KUKA KRL program: MyProgram_093().src

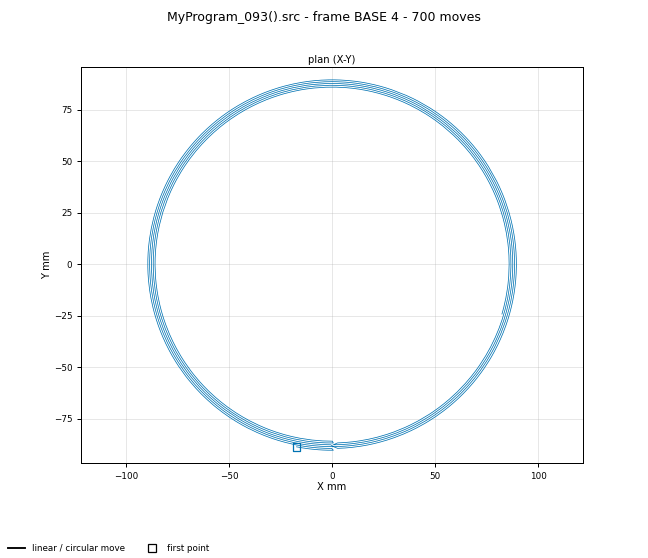
[picture p0: tool path of MyProgram_093().src in frame BASE 4, 700 of 700 moves have a stored position in this frame; points joined in program order, loops and branches not executed]
&ACCESS RVP
&REL 1
&PARAM TEMPLATE = C:\KRC\Roboter\Template\vorgabe
&PARAM EDITMASK = *
DEF MyProgram_093()
; ---- Setting reference (Base) ----
$BASE = BASE_DATA[4]

; --------------------------
; ---- Setting tool (TCP) ----
$TOOL = TOOL_DATA[3]
; --------------------------

$VEL.CP = VEL_APROX_PRINT
Startdeposition()
$VEL.CP = VEL_PRINT
LIN {X -17.2677,Y -88.7195,Z 88,A -105.0819,B 24.9302,C -1.9284,E1 24.9711,E2 190.1577} C_DIS
LIN {X -14.1349,Y -89.2726,Z 88,A -103.3335,B 24.931,C -1.9189,E1 24.9759,E2 188.4301} C_DIS
LIN {X -11.9398,Y -89.5926,Z 88,A -101.7935,B 24.9307,C -1.923,E1 24.9801,E2 186.8791} C_DIS
LIN {X -9.7374,Y -89.8586,Z 88,A -100.3354,B 24.9306,C -1.9245,E1 24.9842,E2 185.4164} C_DIS
LIN {X -6.6492,Y -90.1409,Z 88,A -98.31,B 24.9304,C -1.9264,E1 24.9899,E2 183.3856} C_DIS
LIN {X -4.435,Y -90.2769,Z 88,A -96.9041,B 24.9304,C -1.9265,E1 24.9938,E2 181.9792} C_DIS
LIN {X -2.2182,Y -90.3586,Z 88,A -95.6086,B 24.9307,C -1.923,E1 24.9974,E2 180.6918} C_DIS
LIN {X 0.6077,Y -90.3807,Z 88,A -93.9914,B 24.9311,C -1.9176,E1 25.0019,E2 179.0874} C_DIS
Enddeposition()
LIN {X 0.6077,Y -90.3807,Z 88,A -93.9914,B 24.9311,C -1.9176,E1 25.0019,E2 179.0874} C_DIS
Startdeposition()
$VEL.CP = VEL_PRINT
LIN {X -0.2018,Y -89.5034,Z 88,A -95.2008,B 24.9316,C -1.91,E1 24.9984,E2 180.3149} C_DIS
LIN {X -3.7428,Y -89.4247,Z 88,A -97.2969,B 24.9312,C -1.9153,E1 24.9926,E2 182.3987} C_DIS
LIN {X -6.611,Y -89.26,Z 88,A -99.3502,B 24.9317,C -1.9083,E1 24.9868,E2 184.4693} C_DIS
LIN {X -9.99,Y -88.9447,Z 88,A -101.4992,B 24.9317,C -1.9092,E1 24.9809,E2 186.6173} C_DIS
LIN {X -13.5317,Y -88.4743,Z 88,A -103.6581,B 24.9313,C -1.9139,E1 24.9749,E2 188.7669} C_DIS
LIN {X -16.6632,Y -87.9386,Z 88,A -105.8021,B 24.9315,C -1.911,E1 24.969,E2 190.9198} C_DIS
LIN {X -19.0714,Y -87.4475,Z 88,A -107.3659,B 24.9315,C -1.912,E1 24.9647,E2 192.4831} C_DIS
LIN {X -22.7883,Y -86.5549,Z 88,A -109.8141,B 24.9314,C -1.9133,E1 24.9581,E2 194.9317} C_DIS
LIN {X -26.1366,Y -85.6026,Z 88,A -112.07,B 24.9314,C -1.914,E1 24.9521,E2 197.1898} C_DIS
LIN {X -29.0903,Y -84.6452,Z 88,A -114.4014,B 24.932,C -1.9048,E1 24.9458,E2 199.5475} C_DIS
LIN {X -32.8513,Y -83.2562,Z 88,A -116.3989,B 24.9305,C -1.925,E1 24.9407,E2 201.501} C_DIS
LIN {X -36.4844,Y -81.7299,Z 88,A -119.5254,B 24.9317,C -1.9088,E1 24.9326,E2 204.6734} C_DIS
LIN {X -40.9536,Y -79.5842,Z 88,A -122.2051,B 24.9303,C -1.928,E1 24.926,E2 207.3145} C_DIS
LIN {X -43.6945,Y -78.1126,Z 88,A -124.3723,B 24.9305,C -1.9253,E1 24.9206,E2 209.4945} C_DIS
LIN {X -46.616,Y -76.4052,Z 88,A -126.2873,B 24.9297,C -1.9361,E1 24.9161,E2 211.3894} C_DIS
LIN {X -50.1403,Y -74.14,Z 88,A -129.7875,B 24.9312,C -1.9153,E1 24.9078,E2 214.9507} C_DIS
LIN {X -53.1864,Y -71.9871,Z 88,A -131.414,B 24.9293,C -1.9425,E1 24.9043,E2 216.5181} C_DIS
LIN {X -55.7787,Y -69.9975,Z 88,A -133.5713,B 24.9291,C -1.9443,E1 24.8995,E2 218.6792} C_DIS
LIN {X -57.6179,Y -68.4926,Z 88,A -135.3866,B 24.9296,C -1.9382,E1 24.8956,E2 220.5159} C_DIS
LIN {X -60.6071,Y -65.8603,Z 88,A -137.8417,B 24.929,C -1.9461,E1 24.8905,E2 222.962} C_DIS
LIN {X -63.6381,Y -62.9364,Z 88,A -140.4239,B 24.9283,C -1.9551,E1 24.8854,E2 225.5335} C_DIS
LIN {X -65.9632,Y -60.495,Z 88,A -142.6569,B 24.9282,C -1.9576,E1 24.8811,E2 227.7704} C_DIS
LIN {X -69.4849,Y -56.4149,Z 88,A -146.0739,B 24.9275,C -1.9665,E1 24.8749,E2 231.1817} C_DIS
LIN {X -71.1283,Y -54.3295,Z 88,A -147.9693,B 24.9276,C -1.9647,E1 24.8717,E2 233.0904} C_DIS
LIN {X -74.4966,Y -49.6106,Z 88,A -151.3869,B 24.9263,C -1.9827,E1 24.8663,E2 236.4819} C_DIS
LIN {X -75.9809,Y -47.3044,Z 88,A -153.3686,B 24.9265,C -1.9806,E1 24.8633,E2 238.4788} C_DIS
LIN {X -77.7777,Y -44.2893,Z 88,A -155.6267,B 24.926,C -1.9862,E1 24.8601,E2 240.7353} C_DIS
LIN {X -79.0548,Y -41.9667,Z 88,A -157.3694,B 24.9258,C -1.9894,E1 24.8578,E2 242.4794} C_DIS
LIN {X -80.6854,Y -38.7382,Z 88,A -159.5317,B 24.925,C -2.0004,E1 24.8551,E2 244.6274} C_DIS
LIN {X -82.1108,Y -35.6177,Z 88,A -161.8296,B 24.9247,C -2.0036,E1 24.8525,E2 246.9302} C_DIS
LIN {X -83.3917,Y -32.5064,Z 88,A -164.0572,B 24.9244,C -2.0077,E1 24.8502,E2 249.1605} C_DIS
LIN {X -84.4231,Y -29.7244,Z 88,A -165.8189,B 24.9237,C -2.0172,E1 24.8485,E2 250.9093} C_DIS
LIN {X -85.4184,Y -26.7309,Z 88,A -167.9478,B 24.9235,C -2.0201,E1 24.8467,E2 253.0437} C_DIS
LIN {X -86.2514,Y -23.9112,Z 88,A -169.6906,B 24.9227,C -2.0298,E1 24.8454,E2 254.7735} C_DIS
LIN {X -86.9893,Y -21.0635,Z 88,A -171.7604,B 24.9227,C -2.0301,E1 24.844,E2 256.8545} C_DIS
LIN {X -88.0046,Y -16.3156,Z 88,A -174.9311,B 24.9221,C -2.0379,E1 24.8422,E2 260.0254} C_DIS
LIN {X -88.5955,Y -12.7139,Z 88,A -177.5639,B 24.9222,C -2.0367,E1 24.8411,E2 262.6767} C_DIS
LIN {X -89.16,Y -7.8382,Z 88,A 179.5846,B 24.9208,C -2.0549,E1 24.8403,E2 265.5017} C_DIS
LIN {X -89.3876,Y -4.5587,Z 88,A 177.4493,B 24.9204,C -2.0607,E1 24.8399,E2 267.636} C_DIS
LIN {X -89.4911,Y -1.4707,Z 88,A 175.3618,B 24.9201,C -2.0639,E1 24.8398,E2 269.7285} C_DIS
LIN {X -89.4749,Y 2.2886,Z 88,A 173.034,B 24.9193,C -2.0738,E1 24.8398,E2 272.0467} C_DIS
LIN {X -89.3176,Y 5.7646,Z 88,A 170.7534,B 24.9189,C -2.0795,E1 24.8402,E2 274.3276} C_DIS
LIN {X -89.0787,Y 8.7189,Z 88,A 168.9357,B 24.9183,C -2.0878,E1 24.8407,E2 276.1363} C_DIS
LIN {X -88.6731,Y 12.1676,Z 88,A 165.5912,B 24.9202,C -2.063,E1 24.842,E2 279.5599} C_DIS
LIN {X -87.7877,Y 17.4455,Z 88,A 163.4378,B 24.9165,C -2.1101,E1 24.8431,E2 281.6135} C_DIS
LIN {X -86.6183,Y 22.5416,Z 88,A 159.8021,B 24.9163,C -2.1124,E1 24.8454,E2 285.2653} C_DIS
LIN {X -85.642,Y 26.0098,Z 88,A 157.6135,B 24.9155,C -2.123,E1 24.8471,E2 287.4412} C_DIS
LIN {X -84.9077,Y 28.3119,Z 88,A 155.9613,B 24.9153,C -2.1247,E1 24.8485,E2 289.0986} C_DIS
LIN {X -83.7002,Y 31.7028,Z 88,A 153.6656,B 24.9147,C -2.1321,E1 24.8507,E2 291.3899} C_DIS
LIN {X -82.4438,Y 34.8398,Z 88,A 151.4698,B 24.9143,C -2.1377,E1 24.8531,E2 293.5845} C_DIS
LIN {X -81.0499,Y 37.9703,Z 88,A 149.4534,B 24.9134,C -2.1494,E1 24.8554,E2 295.5839} C_DIS
LIN {X -79.8135,Y 40.5051,Z 88,A 147.599,B 24.913,C -2.1533,E1 24.8577,E2 297.439} C_DIS
LIN {X -78.7808,Y 42.4785,Z 88,A 145.6712,B 24.9139,C -2.1429,E1 24.8603,E2 299.4018} C_DIS
LIN {X -76.5712,Y 46.3429,Z 88,A 143.1007,B 24.9126,C -2.1591,E1 24.8639,E2 301.9469} C_DIS
LIN {X -74.7509,Y 49.2249,Z 88,A 141.0808,B 24.9117,C -2.1699,E1 24.8669,E2 303.9513} C_DIS
LIN {X -72.9491,Y 51.8579,Z 88,A 139.0218,B 24.9113,C -2.175,E1 24.8702,E2 306.0082} C_DIS
LIN {X -70.896,Y 54.631,Z 88,A 136.746,B 24.9109,C -2.179,E1 24.874,E2 308.2855} C_DIS
LIN {X -68.7971,Y 57.2516,Z 88,A 134.6193,B 24.9104,C -2.1852,E1 24.8777,E2 310.4072} C_DIS
LIN {X -66.6997,Y 59.6819,Z 88,A 132.4938,B 24.9102,C -2.1884,E1 24.8817,E2 312.5348} C_DIS
LIN {X -64.9308,Y 61.603,Z 88,A 130.9514,B 24.9095,C -2.1963,E1 24.8846,E2 314.0651} C_DIS
LIN {X -63.432,Y 63.145,Z 88,A 128.789,B 24.9111,C -2.1766,E1 24.889,E2 316.2837} C_DIS
LIN {X -60.7666,Y 65.714,Z 88,A 127.0312,B 24.9092,C -2.2,E1 24.8924,E2 317.9927} C_DIS
LIN {X -58.1889,Y 68.0064,Z 88,A 124.7992,B 24.9089,C -2.2043,E1 24.8971,E2 320.2233} C_DIS
LIN {X -55.9485,Y 69.8629,Z 88,A 122.8516,B 24.9087,C -2.2058,E1 24.9014,E2 322.1746} C_DIS
LIN {X -53.4359,Y 71.8021,Z 88,A 120.9029,B 24.9082,C -2.2125,E1 24.9057,E2 324.1144} C_DIS
LIN {X -50.8147,Y 73.6801,Z 88,A 118.8448,B 24.9078,C -2.2168,E1 24.9104,E2 326.1693} C_DIS
LIN {X -48.2042,Y 75.4133,Z 88,A 116.8196,B 24.9075,C -2.2201,E1 24.9151,E2 328.1933} C_DIS
LIN {X -45.5838,Y 77.0253,Z 88,A 114.7982,B 24.9074,C -2.2221,E1 24.9199,E2 330.2161} C_DIS
LIN {X -42.1374,Y 78.9649,Z 88,A 111.5734,B 24.9087,C -2.2056,E1 24.928,E2 333.4893} C_DIS
LIN {X -38.5937,Y 80.7549,Z 88,A 109.2049,B 24.908,C -2.2148,E1 24.9339,E2 335.8421} C_DIS
LIN {X -35.4902,Y 82.166,Z 88,A 107.6558,B 24.9061,C -2.2371,E1 24.9377,E2 337.3416} C_DIS
LIN {X -32.6192,Y 83.3474,Z 88,A 105.4788,B 24.9064,C -2.2341,E1 24.9434,E2 339.5308} C_DIS
LIN {X -29.7668,Y 84.4082,Z 88,A 103.7025,B 24.9057,C -2.2418,E1 24.948,E2 341.2922} C_DIS
LIN {X -25.866,Y 85.685,Z 88,A 100.9377,B 24.9058,C -2.2406,E1 24.9554,E2 344.0648} C_DIS
LIN {X -23.2236,Y 86.4376,Z 88,A 98.3447,B 24.9078,C -2.2168,E1 24.9626,E2 346.7182} C_DIS
LIN {X -18.8337,Y 87.4993,Z 88,A 96.2593,B 24.9055,C -2.2442,E1 24.9681,E2 348.7413} C_DIS
LIN {X -14.431,Y 88.3326,Z 88,A 93.5704,B 24.9049,C -2.252,E1 24.9754,E2 351.4145} C_DIS
LIN {X -11.5589,Y 88.7535,Z 88,A 91.666,B 24.9049,C -2.2517,E1 24.9807,E2 353.3209} C_DIS
LIN {X -8.7008,Y 89.0803,Z 88,A 89.6908,B 24.9052,C -2.2484,E1 24.9862,E2 355.305} C_DIS
LIN {X -5.2715,Y 89.3482,Z 88,A 87.4703,B 24.9052,C -2.2488,E1 24.9924,E2 357.5256} C_DIS
LIN {X -1.6513,Y 89.4878,Z 88,A 85.3192,B 24.9046,C -2.2548,E1 24.9984,E2 359.6628} C_DIS
LIN {X 1.2208,Y 89.4957,Z 88,A 83.5226,B 24.9045,C -2.2565,E1 25.0034,E2 361.4553} C_DIS
LIN {X 3.9685,Y 89.415,Z 88,A 81.5419,B 24.9051,C -2.2496,E1 25.0089,E2 363.4518} C_DIS
LIN {X 7.649,Y 89.177,Z 88,A 79.1414,B 24.9051,C -2.2482,E1 25.0156,E2 365.8545} C_DIS
LIN {X 11.3103,Y 88.7857,Z 88,A 76.8921,B 24.9049,C -2.2512,E1 25.0218,E2 368.0948} C_DIS
LIN {X 14.1032,Y 88.3859,Z 88,A 75.0274,B 24.9051,C -2.2488,E1 25.027,E2 369.9635} C_DIS
LIN {X 16.6245,Y 87.946,Z 88,A 73.3814,B 24.9052,C -2.2479,E1 25.0315,E2 371.6098} C_DIS
LIN {X 20.2306,Y 87.1867,Z 88,A 71.1863,B 24.9049,C -2.2521,E1 25.0375,E2 373.792} C_DIS
LIN {X 22.8843,Y 86.5293,Z 88,A 69.2148,B 24.9056,C -2.2438,E1 25.0429,E2 375.7802} C_DIS
LIN {X 25.8223,Y 85.698,Z 88,A 66.9153,B 24.9066,C -2.2311,E1 25.0491,E2 378.1057} C_DIS
LIN {X 28.8694,Y 84.7197,Z 88,A 65.256,B 24.9057,C -2.2422,E1 25.0534,E2 379.7357} C_DIS
LIN {X 36.0471,Y 81.9237,Z 88,A 60.3436,B 24.9061,C -2.2378,E1 25.0661,E2 384.6473} C_DIS
LIN {X 39.2906,Y 80.4195,Z 88,A 58.3164,B 24.9056,C -2.2438,E1 25.0712,E2 386.6551} C_DIS
LIN {X 41.6313,Y 79.2315,Z 88,A 56.109,B 24.9072,C -2.2241,E1 25.0767,E2 388.903} C_DIS
LIN {X 47.5385,Y 75.8347,Z 88,A 51.4751,B 24.9085,C -2.2086,E1 25.0879,E2 393.5592} C_DIS
LIN {X 50.7352,Y 73.7354,Z 88,A 49.6306,B 24.9071,C -2.2248,E1 25.0921,E2 395.359} C_DIS
LIN {X 53.557,Y 71.7112,Z 88,A 47.4868,B 24.9072,C -2.2237,E1 25.0969,E2 397.4979} C_DIS
LIN {X 55.8435,Y 69.9463,Z 88,A 45.6499,B 24.9075,C -2.2207,E1 25.1009,E2 399.3351} C_DIS
LIN {X 57.7632,Y 68.3691,Z 88,A 44.2922,B 24.9071,C -2.2257,E1 25.1038,E2 400.6759} C_DIS
LIN {X 60.1768,Y 66.2551,Z 88,A 41.9475,B 24.9082,C -2.2117,E1 25.1087,E2 403.0443} C_DIS
LIN {X 62.7183,Y 63.8534,Z 88,A 39.7767,B 24.9084,C -2.2094,E1 25.1131,E2 405.2116} C_DIS
LIN {X 64.9615,Y 61.5703,Z 88,A 37.6939,B 24.9089,C -2.2038,E1 25.1171,E2 407.2987} C_DIS
LIN {X 66.5632,Y 59.8344,Z 88,A 36.1594,B 24.9092,C -2.1996,E1 25.12,E2 408.8362} C_DIS
LIN {X 68.486,Y 57.6259,Z 88,A 34.2585,B 24.9097,C -2.1944,E1 25.1235,E2 410.7408} C_DIS
LIN {X 70.6649,Y 54.9308,Z 88,A 32.1916,B 24.9097,C -2.1944,E1 25.127,E2 412.7981} C_DIS
LIN {X 72.0544,Y 53.0944,Z 88,A 30.6065,B 24.9103,C -2.1869,E1 25.1297,E2 414.3932} C_DIS
LIN {X 74.1876,Y 50.07,Z 88,A 28.4301,B 24.9103,C -2.1877,E1 25.1331,E2 416.5571} C_DIS
LIN {X 75.8828,Y 47.4615,Z 88,A 26.1245,B 24.9115,C -2.1716,E1 25.1366,E2 418.8891} C_DIS
LIN {X 79.9299,Y 40.2772,Z 88,A 21.0065,B 24.9123,C -2.1629,E1 25.1435,E2 424.0009} C_DIS
LIN {X 81.5034,Y 36.9869,Z 88,A 18.785,B 24.9125,C -2.1603,E1 25.1461,E2 426.2164} C_DIS
LIN {X 82.8611,Y 33.8353,Z 88,A 16.686,B 24.9127,C -2.1575,E1 25.1484,E2 428.3106} C_DIS
LIN {X 84.0143,Y 30.8614,Z 88,A 14.3901,B 24.9139,C -2.1425,E1 25.1507,E2 430.629} C_DIS
LIN {X 85.8827,Y 25.1996,Z 88,A 10.5558,B 24.9149,C -2.1305,E1 25.1539,E2 434.4699} C_DIS
LIN {X 86.8929,Y 21.4584,Z 88,A 8.2472,B 24.9149,C -2.129,E1 25.1555,E2 436.7687} C_DIS
LIN {X 87.6431,Y 18.1519,Z 88,A 6.0741,B 24.9155,C -2.1223,E1 25.1568,E2 438.9451} C_DIS
LIN {X 88.3202,Y 14.5052,Z 88,A 3.9319,B 24.9155,C -2.1231,E1 25.1578,E2 441.0728} C_DIS
LIN {X 88.737,Y 11.6858,Z 88,A 2.1199,B 24.9159,C -2.1178,E1 25.1585,E2 442.8865} C_DIS
LIN {X 89.062,Y 8.8849,Z 88,A 0.3349,B 24.9163,C -2.1128,E1 25.1591,E2 444.6728} C_DIS
LIN {X 89.31,Y 5.8763,Z 88,A -1.6468,B 24.9169,C -2.1049,E1 25.1595,E2 446.6614} C_DIS
LIN {X 89.4643,Y 2.6332,Z 88,A -3.8473,B 24.9178,C -2.094,E1 25.1598,E2 448.8747} C_DIS
LIN {X 89.4981,Y -1.0756,Z 88,A -6.2174,B 24.9184,C -2.0865,E1 25.1598,E2 451.2484} C_DIS
LIN {X 89.3856,Y -4.5956,Z 88,A -8.4623,B 24.9189,C -2.0796,E1 25.1595,E2 453.4961} C_DIS
LIN {X 89.1712,Y -7.7166,Z 88,A -10.4271,B 24.9193,C -2.0745,E1 25.1591,E2 455.4613} C_DIS
LIN {X 88.8268,Y -10.9927,Z 88,A -12.5395,B 24.9198,C -2.0676,E1 25.1584,E2 457.5775} C_DIS
LIN {X 88.3477,Y -14.3402,Z 88,A -14.7309,B 24.9204,C -2.0597,E1 25.1574,E2 459.7745} C_DIS
LIN {X 87.756,Y -17.6022,Z 88,A -16.4946,B 24.92,C -2.0658,E1 25.1565,E2 461.5136} C_DIS
LIN {X 87.0982,Y -20.6136,Z 88,A -18.7695,B 24.9213,C -2.0487,E1 25.1551,E2 463.8155} C_DIS
LIN {X 86.2975,Y -23.7425,Z 88,A -20.7239,B 24.9215,C -2.0463,E1 25.1537,E2 465.7645} C_DIS
LIN {X 85.4502,Y -26.6282,Z 88,A -22.6821,B 24.922,C -2.0391,E1 25.1521,E2 467.7286} C_DIS
LIN {X 84.4861,Y -29.5448,Z 88,A -24.9873,B 24.9234,C -2.021,E1 25.15,E2 470.0635} C_DIS
LIN {X 83.0641,Y -33.3367,Z 88,A -27.0152,B 24.9225,C -2.033,E1 25.148,E2 472.0517} C_DIS
LIN {X 81.6672,Y -36.6235,Z 88,A -29.3937,B 24.9233,C -2.0228,E1 25.1454,E2 474.4412} C_DIS
LIN {X 80.448,Y -39.2321,Z 88,A -31.4259,B 24.9242,C -2.0106,E1 25.1429,E2 476.4914} C_DIS
LIN {X 78.7402,Y -42.5534,Z 88,A -33.5786,B 24.9241,C -2.0121,E1 25.1401,E2 478.6293} C_DIS
LIN {X 77.4747,Y -44.8165,Z 88,A -35.2901,B 24.9246,C -2.0054,E1 25.1377,E2 480.3476} C_DIS
LIN {X 76.2837,Y -46.8149,Z 88,A -37.6884,B 24.9273,C -1.9692,E1 25.1341,E2 482.8192} C_DIS
LIN {X 73.7357,Y -50.7348,Z 88,A -39.8088,B 24.9256,C -1.9915,E1 25.1309,E2 484.8766} C_DIS
LIN {X 72.3535,Y -52.6859,Z 88,A -41.317,B 24.9259,C -1.9881,E1 25.1284,E2 486.3854} C_DIS
LIN {X 70.2113,Y -55.5082,Z 88,A -43.4754,B 24.9261,C -1.9859,E1 25.1247,E2 488.5388} C_DIS
LIN {X 68.3715,Y -57.7604,Z 88,A -45.5353,B 24.9269,C -1.9741,E1 25.121,E2 490.6172} C_DIS
LIN {X 66.2879,Y -60.1411,Z 88,A -47.5453,B 24.9273,C -1.9695,E1 25.1173,E2 492.6292} C_DIS
LIN {X 63.6878,Y -62.886,Z 88,A -49.7628,B 24.9272,C -1.9706,E1 25.113,E2 494.8343} C_DIS
LIN {X 61.5704,Y -64.9615,Z 88,A -51.7185,B 24.9277,C -1.9641,E1 25.1091,E2 496.7974} C_DIS
LIN {X 59.1043,Y -67.2128,Z 88,A -53.608,B 24.9274,C -1.9678,E1 25.1052,E2 498.6705} C_DIS
LIN {X 56.6616,Y -69.2849,Z 88,A -55.8817,B 24.9283,C -1.9554,E1 25.1003,E2 500.9646} C_DIS
LIN {X 54.0322,Y -71.3542,Z 88,A -58.0083,B 24.9286,C -1.9514,E1 25.0956,E2 503.0931} C_DIS
LIN {X 50.5398,Y -73.8695,Z 88,A -60.7922,B 24.9291,C -1.9448,E1 25.0892,E2 505.8829} C_DIS
LIN {X 47.5934,Y -75.8003,Z 88,A -63.0457,B 24.9294,C -1.9405,E1 25.0839,E2 508.1392} C_DIS
LIN {X 45.0862,Y -77.3189,Z 88,A -65.7477,B 24.9317,C -1.9089,E1 25.0772,E2 510.9076} C_DIS
LIN {X 41.0599,Y -79.5299,Z 88,A -67.8581,B 24.93,C -1.9321,E1 25.0722,E2 512.9572} C_DIS
LIN {X 38.2002,Y -80.9429,Z 88,A -69.9562,B 24.9304,C -1.927,E1 25.0669,E2 515.0621} C_DIS
LIN {X 34.4692,Y -82.6,Z 88,A -72.711,B 24.931,C -1.9183,E1 25.0597,E2 517.8307} C_DIS
LIN {X 30.2241,Y -84.2467,Z 88,A -75.53,B 24.931,C -1.9177,E1 25.0524,E2 520.6453} C_DIS
LIN {X 26.6354,Y -85.448,Z 88,A -77.7297,B 24.9307,C -1.9223,E1 25.0466,E2 522.8299} C_DIS
LIN {X 23.5822,Y -86.3407,Z 88,A -79.7732,B 24.9309,C -1.9198,E1 25.0411,E2 524.876} C_DIS
LIN {X 20.5418,Y -87.1148,Z 88,A -81.8168,B 24.9311,C -1.9166,E1 25.0355,E2 526.9241} C_DIS
LIN {X 17.3379,Y -87.8087,Z 88,A -83.9793,B 24.9314,C -1.9127,E1 25.0296,E2 529.0933} C_DIS
LIN {X 13.9414,Y -88.4109,Z 88,A -86.2356,B 24.9317,C -1.9094,E1 25.0234,E2 531.355} C_DIS
LIN {X 9.9536,Y -88.949,Z 88,A -88.7751,B 24.9317,C -1.909,E1 25.0163,E2 533.8935} C_DIS
LIN {X 6.3255,Y -89.2797,Z 88,A -91.0284,B 24.9316,C -1.9105,E1 25.0101,E2 536.1421} C_DIS
LIN {X 2.7078,Y -89.462,Z 88,A -93.338,B 24.9316,C -1.91,E1 25.0036,E2 538.4523} C_DIS
LIN {X 2.7078,Y -89.462,Z 88,A -93.338,B 24.9316,C -1.91,E1 25.0036,E2 538.4523} C_DIS
Enddeposition()
LIN {X 0.6005,Y -88.6192,Z 88,A -94.3434,B 24.9297,C -1.9363,E1 25.001,E2 539.3951} C_DIS
Startdeposition()
$VEL.CP = VEL_PRINT
LIN {X 3.1976,Y -88.5651,Z 88,A -91.8412,B 24.9277,C -1.9639,E1 25.0082,E2 536.828} C_DIS
LIN {X 6.3185,Y -88.397,Z 88,A -89.953,B 24.9279,C -1.9603,E1 25.0134,E2 534.9489} C_DIS
LIN {X 9.8209,Y -88.0774,Z 88,A -87.6368,B 24.9278,C -1.963,E1 25.0198,E2 532.628} C_DIS
LIN {X 14.6258,Y -87.4067,Z 88,A -84.7926,B 24.9283,C -1.9554,E1 25.0276,E2 529.8042} C_DIS
LIN {X 19.3354,Y -86.4881,Z 88,A -81.6865,B 24.9281,C -1.9582,E1 25.0362,E2 526.6955} C_DIS
LIN {X 22.1817,Y -85.8011,Z 88,A -79.5804,B 24.9274,C -1.9673,E1 25.0419,E2 524.5709} C_DIS
LIN {X 25.7596,Y -84.7971,Z 88,A -76.3175,B 24.925,C -1.9994,E1 25.0508,E2 521.2377} C_DIS
LIN {X 30.1765,Y -83.3262,Z 88,A -74.2258,B 24.9271,C -1.9718,E1 25.0561,E2 519.2157} C_DIS
LIN {X 35.5253,Y -81.1899,Z 88,A -70.92,B 24.9278,C -1.9628,E1 25.0646,E2 515.9388} C_DIS
LIN {X 37.4237,Y -80.3325,Z 88,A -69.1799,B 24.9266,C -1.9783,E1 25.0691,E2 514.1663} C_DIS
LIN {X 40.4221,Y -78.8663,Z 88,A -66.7416,B 24.9256,C -1.9915,E1 25.0753,E2 511.7033} C_DIS
LIN {X 45.3685,Y -76.1291,Z 88,A -63.4252,B 24.926,C -1.9863,E1 25.0833,E2 508.4092} C_DIS
LIN {X 47.4501,Y -74.8504,Z 88,A -61.8572,B 24.9258,C -1.9889,E1 25.087,E2 506.8401} C_DIS
LIN {X 49.9456,Y -73.2078,Z 88,A -59.1269,B 24.9234,C -2.0207,E1 25.0934,E2 504.0438} C_DIS
LIN {X 53.3367,Y -70.7747,Z 88,A -57.6129,B 24.9261,C -1.9848,E1 25.0966,E2 502.62} C_DIS
LIN {X 55.22,Y -69.316,Z 88,A -55.1386,B 24.9234,C -2.0209,E1 25.1022,E2 500.0697} C_DIS
LIN {X 57.8911,Y -67.1025,Z 88,A -53.6062,B 24.9249,C -2.0009,E1 25.1054,E2 498.5904} C_DIS
LIN {X 60.9394,Y -64.3453,Z 88,A -51.0838,B 24.9249,C -2.0024,E1 25.1105,E2 496.0748} C_DIS
LIN {X 62.5913,Y -62.7404,Z 88,A -49.2844,B 24.9237,C -2.0168,E1 25.1142,E2 494.2488} C_DIS
LIN {X 65.7563,Y -59.4147,Z 88,A -46.6063,B 24.9239,C -2.014,E1 25.1192,E2 491.589} C_DIS
LIN {X 69.0689,Y -55.5288,Z 88,A -43.1583,B 24.9229,C -2.0277,E1 25.1255,E2 488.1245} C_DIS
LIN {X 71.9735,Y -51.7082,Z 88,A -39.9436,B 24.922,C -2.0401,E1 25.1309,E2 484.896} C_DIS
LIN {X 75.1163,Y -47.0254,Z 88,A -36.3964,B 24.9214,C -2.0467,E1 25.1363,E2 481.3508} C_DIS
LIN {X 77.8286,Y -42.386,Z 88,A -33.1753,B 24.9214,C -2.0477,E1 25.1408,E2 478.144} C_DIS
LIN {X 78.9906,Y -40.1789,Z 88,A -31.2792,B 24.9202,C -2.0626,E1 25.1432,E2 476.2229} C_DIS
LIN {X 81.9041,Y -33.8495,Z 88,A -27.0431,B 24.9199,C -2.0664,E1 25.1481,E2 472.0006} C_DIS
LIN {X 84.0198,Y -28.1874,Z 88,A -22.919,B 24.9184,C -2.0862,E1 25.152,E2 467.853} C_DIS
LIN {X 85.0659,Y -24.8548,Z 88,A -20.6751,B 24.9179,C -2.0927,E1 25.1538,E2 465.6065} C_DIS
LIN {X 85.9492,Y -21.6053,Z 88,A -17.8783,B 24.9156,C -2.122,E1 25.1558,E2 462.7568} C_DIS
LIN {X 86.8022,Y -17.8664,Z 88,A -16.1775,B 24.9172,C -2.1018,E1 25.1568,E2 461.1136} C_DIS
LIN {X 87.6132,Y -13.3345,Z 88,A -13.2637,B 24.9166,C -2.109,E1 25.1581,E2 458.1998} C_DIS
LIN {X 88.0143,Y -10.36,Z 88,A -11.2366,B 24.9158,C -2.1183,E1 25.1589,E2 456.1626} C_DIS
LIN {X 88.3956,Y -6.3391,Z 88,A -8.6111,B 24.9151,C -2.1272,E1 25.1595,E2 453.5317} C_DIS
LIN {X 88.5626,Y -3.2725,Z 88,A -6.6765,B 24.9148,C -2.1317,E1 25.1597,E2 451.5979} C_DIS
LIN {X 88.6216,Y -0.3011,Z 88,A -4.8061,B 24.9144,C -2.1361,E1 25.1597,E2 449.7284} C_DIS
LIN {X 88.5857,Y 2.5396,Z 88,A -2.9037,B 24.9138,C -2.1443,E1 25.1597,E2 447.8179} C_DIS
LIN {X 88.389,Y 6.4378,Z 88,A -0.4083,B 24.9132,C -2.1513,E1 25.1592,E2 445.3209} C_DIS
LIN {X 88.1096,Y 9.5199,Z 88,A 1.6134,B 24.9126,C -2.1584,E1 25.1587,E2 443.2944} C_DIS
LIN {X 87.727,Y 12.5624,Z 88,A 3.6569,B 24.9119,C -2.1668,E1 25.1579,E2 441.243} C_DIS
LIN {X 87.1772,Y 15.9387,Z 88,A 6.4505,B 24.9097,C -2.1946,E1 25.1565,E2 438.4002} C_DIS
LIN {X 86.3752,Y 19.8288,Z 88,A 7.8866,B 24.9123,C -2.162,E1 25.1557,E2 437.0494} C_DIS
LIN {X 85.0889,Y 24.7756,Z 88,A 11.521,B 24.9106,C -2.1837,E1 25.1531,E2 433.3846} C_DIS
LIN {X 83.447,Y 29.845,Z 88,A 15.0329,B 24.9095,C -2.1963,E1 25.15,E2 429.8629} C_DIS
LIN {X 82.2935,Y 32.8922,Z 88,A 17.1699,B 24.9089,C -2.2035,E1 25.1478,E2 427.7208} C_DIS
LIN {X 80.9442,Y 36.0832,Z 88,A 19.372,B 24.9085,C -2.2085,E1 25.1453,E2 425.5188} C_DIS
LIN {X 79.36,Y 39.444,Z 88,A 21.3779,B 24.9091,C -2.2013,E1 25.1429,E2 423.5408} C_DIS
LIN {X 76.9546,Y 43.9532,Z 88,A 25.0166,B 24.9074,C -2.222,E1 25.1381,E2 419.8722} C_DIS
LIN {X 74.8134,Y 47.5076,Z 88,A 27.6637,B 24.9069,C -2.2277,E1 25.1342,E2 417.2251} C_DIS
LIN {X 72.9779,Y 50.2812,Z 88,A 29.7743,B 24.9066,C -2.2318,E1 25.1309,E2 415.1153} C_DIS
LIN {X 70.7046,Y 53.43,Z 88,A 31.9984,B 24.9069,C -2.228,E1 25.1272,E2 412.9109} C_DIS
LIN {X 69.3139,Y 55.2227,Z 88,A 33.9602,B 24.9051,C -2.2487,E1 25.1238,E2 410.9093} C_DIS
LIN {X 66.9386,Y 58.0788,Z 88,A 36.7117,B 24.9036,C -2.2664,E1 25.1187,E2 408.1284} C_DIS
LIN {X 64.6016,Y 60.6669,Z 88,A 38.2208,B 24.9054,C -2.2455,E1 25.116,E2 406.6754} C_DIS
LIN {X 62.789,Y 62.5421,Z 88,A 40.094,B 24.9046,C -2.2555,E1 25.1123,E2 404.7865} C_DIS
LIN {X 60.2687,Y 64.975,Z 88,A 42.9043,B 24.9026,C -2.279,E1 25.1064,E2 401.9321} C_DIS
LIN {X 57.6465,Y 67.311,Z 88,A 44.6105,B 24.9038,C -2.264,E1 25.1029,E2 400.2682} C_DIS
LIN {X 54.3178,Y 70.0249,Z 88,A 47.3549,B 24.9035,C -2.268,E1 25.0969,E2 397.5246} C_DIS
LIN {X 51.4091,Y 72.1869,Z 88,A 49.6351,B 24.9033,C -2.2699,E1 25.0918,E2 395.2481} C_DIS
LIN {X 47.1286,Y 75.0518,Z 88,A 53.4368,B 24.9015,C -2.2911,E1 25.0828,E2 391.4084} C_DIS
LIN {X 43.6175,Y 77.1464,Z 88,A 55.6468,B 24.9025,C -2.2802,E1 25.0776,E2 389.2309} C_DIS
LIN {X 40.6525,Y 78.7486,Z 88,A 57.8876,B 24.902,C -2.2852,E1 25.072,E2 386.9848} C_DIS
LIN {X 37.0071,Y 80.5264,Z 88,A 60.4801,B 24.9018,C -2.2873,E1 25.0655,E2 384.394} C_DIS
LIN {X 31.7991,Y 82.7212,Z 88,A 64.1364,B 24.9015,C -2.2911,E1 25.056,E2 380.737} C_DIS
LIN {X 29.423,Y 83.5951,Z 88,A 65.6981,B 24.9016,C -2.2901,E1 25.0519,E2 379.1809} C_DIS
LIN {X 24.1408,Y 85.2705,Z 88,A 69.7711,B 24.9,C -2.3089,E1 25.0409,E2 375.0703} C_DIS
LIN {X 21.0041,Y 86.0968,Z 88,A 71.3222,B 24.9014,C -2.2922,E1 25.0369,E2 373.5614} C_DIS
LIN {X 15.6068,Y 87.2369,Z 88,A 74.9764,B 24.901,C -2.2966,E1 25.0268,E2 369.9012} C_DIS
LIN {X 11.7881,Y 87.835,Z 88,A 77.1693,B 24.9018,C -2.2873,E1 25.0208,E2 367.7322} C_DIS
LIN {X 9.5705,Y 88.1043,Z 88,A 78.9504,B 24.9009,C -2.2984,E1 25.0158,E2 365.926} C_DIS
LIN {X 6.2427,Y 88.4021,Z 88,A 81.1283,B 24.9009,C -2.2991,E1 25.0098,E2 363.7476} C_DIS
LIN {X 2.3495,Y 88.5915,Z 88,A 83.4367,B 24.9014,C -2.2922,E1 25.0034,E2 361.4564} C_DIS
LIN {X -0.1745,Y 88.6225,Z 88,A 85.2253,B 24.901,C -2.2969,E1 24.9983,E2 359.6567} C_DIS
LIN {X -3.6649,Y 88.5462,Z 88,A 87.7066,B 24.9005,C -2.3034,E1 24.9914,E2 357.1595} C_DIS
LIN {X -10.0171,Y 88.0544,Z 88,A 91.2693,B 24.9022,C -2.2838,E1 24.9816,E2 353.6418} C_DIS
LIN {X -13.6275,Y 87.5679,Z 88,A 94.9307,B 24.8987,C -2.3235,E1 24.9712,E2 349.8826} C_DIS
LIN {X -18.4947,Y 86.6715,Z 88,A 96.8982,B 24.9023,C -2.282,E1 24.9661,E2 348.0116} C_DIS
LIN {X -21.7786,Y 85.9047,Z 88,A 99.8311,B 24.9005,C -2.3035,E1 24.958,E2 345.0237} C_DIS
LIN {X -24.9453,Y 85.0391,Z 88,A 101.3757,B 24.9022,C -2.2832,E1 24.954,E2 343.5249} C_DIS
LIN {X -28.7742,Y 83.8219,Z 88,A 103.8995,B 24.9027,C -2.2778,E1 24.9473,E2 341.0092} C_DIS
LIN {X -31.096,Y 82.9878,Z 88,A 105.6591,B 24.9024,C -2.2808,E1 24.9426,E2 339.2387} C_DIS
LIN {X -33.9993,Y 81.8418,Z 88,A 108.0129,B 24.9018,C -2.2884,E1 24.9365,E2 336.8618} C_DIS
LIN {X -38.3697,Y 79.885,Z 88,A 111.0485,B 24.9023,C -2.2818,E1 24.9288,E2 333.8342} C_DIS
LIN {X -42.8624,Y 77.5681,Z 88,A 114.8834,B 24.9013,C -2.2937,E1 24.9193,E2 329.9602} C_DIS
LIN {X -46.5883,Y 75.3894,Z 88,A 116.9303,B 24.9037,C -2.2658,E1 24.9146,E2 327.9732} C_DIS
LIN {X -48.9076,Y 73.9047,Z 88,A 118.5389,B 24.9044,C -2.2573,E1 24.9109,E2 326.3799} C_DIS
LIN {X -51.4369,Y 72.1671,Z 88,A 120.616,B 24.9045,C -2.2561,E1 24.9061,E2 324.2984} C_DIS
LIN {X -55.4186,Y 69.1582,Z 88,A 124.1303,B 24.9044,C -2.2579,E1 24.8983,E2 320.767} C_DIS
LIN {X -58.7457,Y 66.3553,Z 88,A 126.7914,B 24.9053,C -2.2471,E1 24.8927,E2 318.1213} C_DIS
LIN {X -61.9476,Y 63.375,Z 88,A 129.7511,B 24.9055,C -2.2444,E1 24.8867,E2 315.1558} C_DIS
LIN {X -65.2039,Y 60.0193,Z 88,A 132.2016,B 24.9075,C -2.22,E1 24.8821,E2 312.7527} C_DIS
LIN {X -66.4278,Y 58.6637,Z 88,A 133.8405,B 24.9067,C -2.2306,E1 24.879,E2 311.0814} C_DIS
LIN {X -68.6219,Y 56.0803,Z 88,A 136.3767,B 24.9063,C -2.2351,E1 24.8744,E2 308.5226} C_DIS
LIN {X -71.6958,Y 52.0927,Z 88,A 139.4807,B 24.9074,C -2.2219,E1 24.8693,E2 305.4353} C_DIS
LIN {X -73.6666,Y 49.268,Z 88,A 141.5971,B 24.9082,C -2.2125,E1 24.866,E2 303.3307} C_DIS
LIN {X -76.3493,Y 44.996,Z 88,A 145.2938,B 24.9079,C -2.2161,E1 24.8606,E2 299.6064} C_DIS
LIN {X -77.9563,Y 42.1505,Z 88,A 146.7267,B 24.91,C -2.1901,E1 24.8587,E2 298.2282} C_DIS
LIN {X -79.1607,Y 39.8462,Z 88,A 149.0221,B 24.909,C -2.203,E1 24.8558,E2 295.8895} C_DIS
LIN {X -80.9994,Y 35.9604,Z 88,A 151.529,B 24.9103,C -2.1868,E1 24.8529,E2 293.4078} C_DIS
LIN {X -82.3203,Y 32.8241,Z 88,A 153.7474,B 24.9108,C -2.1806,E1 24.8505,E2 291.1917} C_DIS
LIN {X -83.6996,Y 29.125,Z 88,A 156.1459,B 24.9118,C -2.1683,E1 24.8483,E2 288.8089} C_DIS
LIN {X -85.0334,Y 24.9646,Z 88,A 159.2168,B 24.9119,C -2.1667,E1 24.8457,E2 285.7244} C_DIS
LIN {X -85.8357,Y 22.0469,Z 88,A 161.6995,B 24.9112,C -2.1759,E1 24.844,E2 283.205} C_DIS
LIN {X -86.7292,Y 18.2215,Z 88,A 163.5304,B 24.9135,C -2.1471,E1 24.8429,E2 281.432} C_DIS
LIN {X -87.6349,Y 13.1919,Z 88,A 166.8697,B 24.9143,C -2.1376,E1 24.8414,E2 278.0956} C_DIS
LIN {X -87.9492,Y 10.909,Z 88,A 169.1556,B 24.9128,C -2.1561,E1 24.8406,E2 275.752} C_DIS
LIN {X -88.357,Y 6.8502,Z 88,A 170.928,B 24.9155,C -2.1224,E1 24.8402,E2 274.0493} C_DIS
LIN {X -88.515,Y 4.3809,Z 88,A 172.6148,B 24.9157,C -2.1198,E1 24.8399,E2 272.3586} C_DIS
LIN {X -88.6099,Y 1.4646,Z 88,A 175.1798,B 24.9146,C -2.1336,E1 24.8398,E2 269.7453} C_DIS
LIN {X -88.5949,Y -2.2272,Z 88,A 177.3391,B 24.9158,C -2.1193,E1 24.8399,E2 267.6071} C_DIS
LIN {X -88.4143,Y -6.0623,Z 88,A 179.3753,B 24.9174,C -2.0984,E1 24.8403,E2 265.6086} C_DIS
LIN {X -88.1608,Y -9.0307,Z 88,A -177.8687,B 24.916,C -2.1166,E1 24.841,E2 262.7926} C_DIS
LIN {X -87.6614,Y -13.0144,Z 88,A -176.0455,B 24.9184,C -2.0858,E1 24.8417,E2 261.032} C_DIS
LIN {X -86.7353,Y -18.1925,Z 88,A -172.6157,B 24.9192,C -2.0761,E1 24.8435,E2 257.6051} C_DIS
LIN {X -86.0801,Y -21.0727,Z 88,A -170.6306,B 24.9195,C -2.0724,E1 24.8448,E2 255.617} C_DIS
LIN {X -85.2066,Y -24.3664,Z 88,A -168.3902,B 24.9199,C -2.0669,E1 24.8464,E2 253.377} C_DIS
LIN {X -84.2051,Y -27.631,Z 88,A -165.8231,B 24.9196,C -2.0709,E1 24.8486,E2 250.7856} C_DIS
LIN {X -83.0371,Y -30.9657,Z 88,A -163.8923,B 24.9209,C -2.0537,E1 24.8505,E2 248.8848} C_DIS
LIN {X -81.965,Y -33.6997,Z 88,A -162.0917,B 24.9216,C -2.0454,E1 24.8523,E2 247.094} C_DIS
LIN {X -79.9876,Y -38.156,Z 88,A -159.1448,B 24.9227,C -2.0304,E1 24.8557,E2 244.1666} C_DIS
LIN {X -78.3965,Y -41.3259,Z 88,A -156.5627,B 24.9225,C -2.0326,E1 24.859,E2 241.5655} C_DIS
LIN {X -76.5397,Y -44.6739,Z 88,A -154.2041,B 24.9233,C -2.0225,E1 24.8622,E2 239.2186} C_DIS
LIN {X -74.6245,Y -47.802,Z 88,A -151.6934,B 24.9234,C -2.0205,E1 24.8659,E2 236.6998} C_DIS
LIN {X -71.9502,Y -51.7403,Z 88,A -148.7029,B 24.9242,C -2.0102,E1 24.8706,E2 233.7192} C_DIS
LIN {X -70.3243,Y -53.9293,Z 88,A -147.0422,B 24.9248,C -2.0029,E1 24.8734,E2 232.068} C_DIS
LIN {X -68.8543,Y -55.7936,Z 88,A -144.6785,B 24.9232,C -2.0242,E1 24.8777,E2 229.6423} C_DIS
LIN {X -66.6635,Y -58.3938,Z 88,A -142.3957,B 24.9233,C -2.0219,E1 24.8819,E2 227.3548} C_DIS
LIN {X -64.1651,Y -61.1306,Z 88,A -139.7503,B 24.9232,C -2.0243,E1 24.887,E2 224.6922} C_DIS
LIN {X -61.0414,Y -64.2495,Z 88,A -137.7014,B 24.9255,C -1.9938,E1 24.891,E2 222.7075} C_DIS
LIN {X -58.5884,Y -66.4935,Z 88,A -134.8793,B 24.9242,C -2.0103,E1 24.897,E2 219.835} C_DIS
LIN {X -55.6128,Y -69.0008,Z 88,A -132.8439,B 24.9257,C -1.9908,E1 24.9013,E2 217.8384} C_DIS
LIN {X -52.6586,Y -71.2815,Z 88,A -130.1043,B 24.9252,C -1.9967,E1 24.9075,E2 215.0749} C_DIS
LIN {X -49.9466,Y -73.2071,Z 88,A -128.1507,B 24.926,C -1.9871,E1 24.912,E2 213.1375} C_DIS
LIN {X -45.8697,Y -75.8277,Z 88,A -125.2486,B 24.9269,C -1.9752,E1 24.9188,E2 210.2546} C_DIS
LIN {X -43.3471,Y -77.2974,Z 88,A -123.4281,B 24.9272,C -1.9705,E1 24.9232,E2 208.44} C_DIS
LIN {X -40.078,Y -79.0422,Z 88,A -121.0995,B 24.9276,C -1.9653,E1 24.929,E2 206.1173} C_DIS
LIN {X -36.2466,Y -80.8706,Z 88,A -118.011,B 24.927,C -1.973,E1 24.9369,E2 203.0028} C_DIS
LIN {X -32.1328,Y -82.5918,Z 88,A -115.4131,B 24.9279,C -1.9611,E1 24.9435,E2 200.4274} C_DIS
LIN {X -27.6276,Y -84.2062,Z 88,A -111.9588,B 24.9272,C -1.97,E1 24.9527,E2 196.9453} C_DIS
LIN {X -23.5781,Y -85.4292,Z 88,A -109.5002,B 24.928,C -1.9593,E1 24.9593,E2 194.5081} C_DIS
LIN {X -18.3389,Y -86.705,Z 88,A -106.1154,B 24.9284,C -1.9543,E1 24.9684,E2 191.1307} C_DIS
LIN {X -14.7938,Y -87.3786,Z 88,A -104.0426,B 24.9291,C -1.9451,E1 24.9741,E2 189.0777} C_DIS
LIN {X -12.3151,Y -87.7622,Z 88,A -102.1573,B 24.9285,C -1.9532,E1 24.9793,E2 187.1714} C_DIS
LIN {X -9.0071,Y -88.1633,Z 88,A -99.8463,B 24.9281,C -1.9581,E1 24.9858,E2 184.8475} C_DIS
LIN {X -5.5391,Y -88.4497,Z 88,A -97.6742,B 24.9283,C -1.9555,E1 24.9918,E2 182.6807} C_DIS
LIN {X -2.1331,Y -88.5976,Z 88,A -95.3672,B 24.928,C -1.9591,E1 24.9983,E2 180.3646} C_DIS
LIN {X 0.6005,Y -88.6192,Z 88,A -94.341,B 24.9298,C -1.9353,E1 25.001,E2 179.3951} C_DIS
Enddeposition()
LIN {X 0.6005,Y -88.6192,Z 88,A -94.341,B 24.9298,C -1.9353,E1 25.001,E2 179.3951} C_DIS
Startdeposition()
$VEL.CP = VEL_PRINT
LIN {X -0.6096,Y -87.7387,Z 88,A -95.5341,B 24.9296,C -1.9376,E1 24.9977,E2 180.5827} C_DIS
LIN {X -4.2859,Y -87.6376,Z 88,A -98.173,B 24.9302,C -1.9297,E1 24.9903,E2 183.2408} C_DIS
LIN {X -9.2552,Y -87.2514,Z 88,A -101.25,B 24.9298,C -1.9356,E1 24.9817,E2 186.3054} C_DIS
LIN {X -12.4437,Y -86.854,Z 88,A -103.1638,B 24.9293,C -1.9418,E1 24.9765,E2 188.2058} C_DIS
LIN {X -16.7811,Y -86.1213,Z 88,A -105.9229,B 24.929,C -1.9463,E1 24.9689,E2 190.957} C_DIS
LIN {X -21.296,Y -85.1179,Z 88,A -109.0723,B 24.9292,C -1.9437,E1 24.9603,E2 194.1167} C_DIS
LIN {X -23.9045,Y -84.4217,Z 88,A -111.7377,B 24.9311,C -1.917,E1 24.953,E2 196.8497} C_DIS
LIN {X -27.9658,Y -83.1647,Z 88,A -113.7984,B 24.9294,C -1.9411,E1 24.9476,E2 198.857} C_DIS
LIN {X -31.2223,Y -81.9978,Z 88,A -115.7213,B 24.9285,C -1.9535,E1 24.9427,E2 200.7544} C_DIS
LIN {X -33.4203,Y -81.1275,Z 88,A -117.3022,B 24.9285,C -1.9538,E1 24.9386,E2 202.338} C_DIS
LIN {X -36.0088,Y -80.0113,Z 88,A -119.5866,B 24.9293,C -1.9423,E1 24.9326,E2 204.6553} C_DIS
LIN {X -39.199,Y -78.4981,Z 88,A -121.9414,B 24.9292,C -1.9435,E1 24.9267,E2 207.0132} C_DIS
LIN {X -42.7653,Y -76.6132,Z 88,A -124.6798,B 24.9292,C -1.9439,E1 24.92,E2 209.7585} C_DIS
LIN {X -45.5368,Y -74.999,Z 88,A -126.8583,B 24.9292,C -1.9445,E1 24.9148,E2 211.9425} C_DIS
LIN {X -51.8736,Y -70.7643,Z 88,A -131.2983,B 24.9273,C -1.9686,E1 24.9047,E2 216.34} C_DIS
LIN {X -54.2264,Y -68.9781,Z 88,A -133.3147,B 24.9273,C -1.9694,E1 24.9002,E2 218.3618} C_DIS
LIN {X -56.3234,Y -67.2771,Z 88,A -135.299,B 24.9275,C -1.9661,E1 24.8959,E2 220.3614} C_DIS
LIN {X -59.1751,Y -64.7827,Z 88,A -137.5071,B 24.9266,C -1.9788,E1 24.8913,E2 222.5481} C_DIS
LIN {X -61.7916,Y -62.2919,Z 88,A -140.0489,B 24.9266,C -1.9783,E1 24.8862,E2 225.1017} C_DIS
LIN {X -64.1792,Y -59.83,Z 88,A -142.4042,B 24.9266,C -1.9798,E1 24.8817,E2 227.4637} C_DIS
LIN {X -68.2756,Y -55.1082,Z 88,A -146.4186,B 24.9257,C -1.9911,E1 24.8744,E2 231.4695} C_DIS
LIN {X -70.363,Y -52.4177,Z 88,A -148.8316,B 24.9257,C -1.991,E1 24.8703,E2 233.8944} C_DIS
LIN {X -73.1836,Y -48.4006,Z 88,A -151.7622,B 24.9245,C -2.007,E1 24.8658,E2 236.8012} C_DIS
LIN {X -75.1832,Y -45.2336,Z 88,A -154.5769,B 24.9248,C -2.0027,E1 24.8616,E2 239.6405} C_DIS
LIN {X -77.2734,Y -41.5616,Z 88,A -156.8588,B 24.9232,C -2.0239,E1 24.8586,E2 241.884} C_DIS
LIN {X -78.5736,Y -39.0467,Z 88,A -158.6559,B 24.9227,C -2.0304,E1 24.8563,E2 243.6751} C_DIS
LIN {X -79.3704,Y -37.4006,Z 88,A -160.643,B 24.9242,C -2.0111,E1 24.8539,E2 245.719} C_DIS
LIN {X -80.7637,Y -34.2888,Z 88,A -162.3162,B 24.9225,C -2.0332,E1 24.8521,E2 247.3489} C_DIS
LIN {X -81.9554,Y -31.3344,Z 88,A -164.107,B 24.9214,C -2.0475,E1 24.8502,E2 249.1156} C_DIS
LIN {X -83.379,Y -27.3221,Z 88,A -167.2888,B 24.9216,C -2.0442,E1 24.8473,E2 252.3233} C_DIS
LIN {X -84.4348,Y -23.8582,Z 88,A -169.652,B 24.9211,C -2.0513,E1 24.8454,E2 254.683} C_DIS
LIN {X -85.3034,Y -20.539,Z 88,A -171.8697,B 24.9205,C -2.0588,E1 24.8439,E2 256.8959} C_DIS
LIN {X -86.0025,Y -17.3807,Z 88,A -174.1193,B 24.9203,C -2.0614,E1 24.8426,E2 259.1525} C_DIS
LIN {X -86.6665,Y -13.691,Z 88,A -177.3679,B 24.9214,C -2.0467,E1 24.8412,E2 262.4555} C_DIS
LIN {X -87.261,Y -9.163,Z 88,A -179.4914,B 24.9189,C -2.0801,E1 24.8405,E2 264.5122} C_DIS
LIN {X -87.6903,Y -2.9908,Z 88,A 176.6064,B 24.9176,C -2.0968,E1 24.8399,E2 268.3979} C_DIS
LIN {X -87.7245,Y 1.6921,Z 88,A 173.7861,B 24.9162,C -2.1132,E1 24.8399,E2 271.1959} C_DIS
LIN {X -87.4691,Y 6.9,Z 88,A 169.4108,B 24.9175,C -2.0969,E1 24.8406,E2 275.6365} C_DIS
LIN {X -87.1355,Y 10.2883,Z 88,A 167.8344,B 24.9155,C -2.1221,E1 24.841,E2 277.1623} C_DIS
LIN {X -86.5789,Y 14.2336,Z 88,A 164.975,B 24.9155,C -2.1232,E1 24.8422,E2 280.0361} C_DIS
LIN {X -85.7879,Y 18.411,Z 88,A 161.81,B 24.9156,C -2.1211,E1 24.844,E2 283.2247} C_DIS
LIN {X -85.0531,Y 21.5522,Z 88,A 160.4936,B 24.9133,C -2.1499,E1 24.8448,E2 284.4801} C_DIS
LIN {X -84.1782,Y 24.7492,Z 88,A 158.3657,B 24.9127,C -2.1577,E1 24.8464,E2 286.6017} C_DIS
LIN {X -83.1615,Y 27.9753,Z 88,A 155.8397,B 24.9128,C -2.1556,E1 24.8486,E2 289.1473} C_DIS
LIN {X -82.1409,Y 30.8443,Z 88,A 153.838,B 24.9124,C -2.1613,E1 24.8505,E2 291.1466} C_DIS
LIN {X -81.0042,Y 33.7182,Z 88,A 151.7044,B 24.9122,C -2.1642,E1 24.8527,E2 293.2853} C_DIS
LIN {X -78.3737,Y 39.45,Z 88,A 147.521,B 24.9113,C -2.1746,E1 24.8577,E2 297.4666} C_DIS
LIN {X -77.1318,Y 41.8226,Z 88,A 145.4474,B 24.9116,C -2.1705,E1 24.8605,E2 299.5608} C_DIS
LIN {X -74.3487,Y 46.5911,Z 88,A 142.0652,B 24.9103,C -2.1871,E1 24.8653,E2 302.921} C_DIS
LIN {X -72.9383,Y 48.772,Z 88,A 140.2466,B 24.9102,C -2.1883,E1 24.8682,E2 304.7459} C_DIS
LIN {X -69.9002,Y 53.0338,Z 88,A 136.2971,B 24.9107,C -2.1825,E1 24.8748,E2 308.7282} C_DIS
LIN {X -67.3548,Y 56.23,Z 88,A 134.3029,B 24.9085,C -2.2085,E1 24.8782,E2 310.6696} C_DIS
LIN {X -65.4833,Y 58.3987,Z 88,A 131.8546,B 24.9095,C -2.1967,E1 24.8829,E2 313.1568} C_DIS
LIN {X -62.9323,Y 61.1399,Z 88,A 130.006,B 24.9076,C -2.2197,E1 24.8863,E2 314.9587} C_DIS
LIN {X -60.434,Y 63.6095,Z 88,A 127.6578,B 24.9073,C -2.2236,E1 24.891,E2 317.3074} C_DIS
LIN {X -57.8236,Y 65.9917,Z 88,A 125.2081,B 24.9072,C -2.2247,E1 24.8962,E2 319.7642} C_DIS
LIN {X -54.8887,Y 68.4535,Z 88,A 122.6802,B 24.9068,C -2.2294,E1 24.9016,E2 322.2904} C_DIS
LIN {X -50.6341,Y 71.6575,Z 88,A 119.5689,B 24.9053,C -2.2472,E1 24.9085,E2 325.3703} C_DIS
LIN {X -47.8653,Y 73.5352,Z 88,A 117.1125,B 24.9056,C -2.2435,E1 24.9143,E2 327.8437} C_DIS
LIN {X -43.1438,Y 76.4018,Z 88,A 113.8017,B 24.9043,C -2.2587,E1 24.9222,E2 331.1283} C_DIS
LIN {X -39.0491,Y 78.5724,Z 88,A 110.491,B 24.9046,C -2.2553,E1 24.9304,E2 334.4563} C_DIS
LIN {X -33.8089,Y 80.9659,Z 88,A 106.7396,B 24.9041,C -2.2611,E1 24.94,E2 338.2028} C_DIS
LIN {X -30.4631,Y 82.2838,Z 88,A 104.4019,B 24.9038,C -2.2646,E1 24.946,E2 340.5373} C_DIS
LIN {X -27.5739,Y 83.2958,Z 88,A 102.2785,B 24.9039,C -2.2633,E1 24.9517,E2 342.6678} C_DIS
LIN {X -24.3318,Y 84.3006,Z 88,A 99.0931,B 24.9061,C -2.2368,E1 24.9604,E2 345.9213} C_DIS
LIN {X -19.2518,Y 85.6042,Z 88,A 95.2934,B 24.9068,C -2.2287,E1 24.9708,E2 349.745} C_DIS
LIN {X -12.9306,Y 86.7841,Z 88,A 92.7636,B 24.9023,C -2.282,E1 24.9775,E2 352.1506} C_DIS
LIN {X -9.433,Y 87.2324,Z 88,A 89.9854,B 24.9034,C -2.2687,E1 24.9853,E2 354.9621} C_DIS
LIN {X -3.4208,Y 87.6748,Z 88,A 86.2704,B 24.9027,C -2.2771,E1 24.9956,E2 358.6584} C_DIS
LIN {X -0.2311,Y 87.741,Z 88,A 84.2075,B 24.9027,C -2.2782,E1 25.0013,E2 360.7187} C_DIS
LIN {X 3.7033,Y 87.6626,Z 88,A 81.3283,B 24.9034,C -2.2689,E1 25.0094,E2 363.6195} C_DIS
LIN {X 7.9693,Y 87.3782,Z 88,A 78.8681,B 24.9026,C -2.2791,E1 25.0162,E2 366.0543} C_DIS
LIN {X 10.5888,Y 87.1003,Z 88,A 76.6376,B 24.9039,C -2.2627,E1 25.0225,E2 368.3218} C_DIS
LIN {X 13.8516,Y 86.6417,Z 88,A 75.1805,B 24.9021,C -2.284,E1 25.0264,E2 369.7272} C_DIS
LIN {X 17.3037,Y 86.0175,Z 88,A 72.6298,B 24.9029,C -2.2748,E1 25.0334,E2 372.2966} C_DIS
LIN {X 19.6318,Y 85.5164,Z 88,A 70.3832,B 24.9048,C -2.2521,E1 25.0397,E2 374.594} C_DIS
LIN {X 23.6589,Y 84.4913,Z 88,A 68.0371,B 24.904,C -2.2619,E1 25.0459,E2 376.9129} C_DIS
LIN {X 27.9213,Y 83.1797,Z 88,A 65.5797,B 24.903,C -2.2742,E1 25.0523,E2 379.3367} C_DIS
LIN {X 30.4051,Y 82.305,Z 88,A 63.4495,B 24.9042,C -2.2594,E1 25.058,E2 381.4975} C_DIS
LIN {X 35.0821,Y 80.422,Z 88,A 60.661,B 24.9031,C -2.2723,E1 25.0651,E2 384.2491} C_DIS
LIN {X 38.5825,Y 78.8037,Z 88,A 58.1173,B 24.9035,C -2.2685,E1 25.0715,E2 386.7952} C_DIS
LIN {X 40.734,Y 77.7124,Z 88,A 56.3975,B 24.904,C -2.2617,E1 25.0758,E2 388.5263} C_DIS
LIN {X 43.194,Y 76.3737,Z 88,A 54.5065,B 24.9044,C -2.2571,E1 25.0804,E2 390.4226} C_DIS
LIN {X 49.457,Y 72.4745,Z 88,A 49.9462,B 24.9044,C -2.2582,E1 25.0912,E2 394.9656} C_DIS
LIN {X 52.7609,Y 70.1052,Z 88,A 46.6667,B 24.9065,C -2.2329,E1 25.0986,E2 398.2932} C_DIS
LIN {X 55.3667,Y 68.0662,Z 88,A 44.9565,B 24.9055,C -2.2438,E1 25.1023,E2 399.9712} C_DIS
LIN {X 60.711,Y 63.3457,Z 88,A 40.3911,B 24.9061,C -2.2376,E1 25.1118,E2 404.533} C_DIS
LIN {X 62.5376,Y 61.5428,Z 88,A 37.6997,B 24.9092,C -2.2002,E1 25.1172,E2 407.3013} C_DIS
LIN {X 65.9373,Y 57.8859,Z 88,A 35.4879,B 24.9069,C -2.2279,E1 25.1211,E2 409.4378} C_DIS
LIN {X 69.2494,Y 53.8807,Z 88,A 31.4266,B 24.9094,C -2.1974,E1 25.1283,E2 413.5523} C_DIS
LIN {X 71.5175,Y 50.8304,Z 88,A 29.5484,B 24.9082,C -2.2116,E1 25.1313,E2 415.3877} C_DIS
LIN {X 73.3561,Y 48.139,Z 88,A 27.7901,B 24.9076,C -2.2189,E1 25.134,E2 417.1202} C_DIS
LIN {X 74.7375,Y 45.967,Z 88,A 25.7731,B 24.909,C -2.203,E1 25.137,E2 419.1645} C_DIS
LIN {X 75.9302,Y 43.9675,Z 88,A 24.2917,B 24.9092,C -2.2003,E1 25.1391,E2 420.6446} C_DIS
LIN {X 78.1777,Y 39.8335,Z 88,A 21.8212,B 24.9082,C -2.2127,E1 25.1424,E2 423.0729} C_DIS
LIN {X 79.5391,Y 37.0402,Z 88,A 19.2712,B 24.9101,C -2.189,E1 25.1455,E2 425.6651} C_DIS
LIN {X 80.9009,Y 33.9634,Z 88,A 17.0849,B 24.9106,C -2.1831,E1 25.1479,E2 427.8535} C_DIS
LIN {X 82.1829,Y 30.7336,Z 88,A 14.752,B 24.9113,C -2.1743,E1 25.1503,E2 430.1941} C_DIS
LIN {X 83.8233,Y 25.9251,Z 88,A 11.3316,B 24.9124,C -2.1609,E1 25.1533,E2 433.6268} C_DIS
LIN {X 85.1726,Y 21.0748,Z 88,A 8.5605,B 24.9118,C -2.1688,E1 25.1553,E2 436.3632} C_DIS
LIN {X 86.3364,Y 15.636,Z 88,A 4.8703,B 24.9129,C -2.1555,E1 25.1574,E2 440.0633} C_DIS
LIN {X 86.9463,Y 11.7922,Z 88,A 2.0598,B 24.9143,C -2.1382,E1 25.1586,E2 442.8983} C_DIS
LIN {X 87.3442,Y 8.3376,Z 88,A -0.1687,B 24.9147,C -2.1325,E1 25.1592,E2 445.127} C_DIS
LIN {X 87.6387,Y 4.2604,Z 88,A -3.0951,B 24.9161,C -2.115,E1 25.1597,E2 448.0772} C_DIS
LIN {X 87.7414,Y 0.1069,Z 88,A -5.513,B 24.916,C -2.1167,E1 25.1597,E2 450.4769} C_DIS
LIN {X 87.6817,Y -3.2579,Z 88,A -7.4755,B 24.9159,C -2.1178,E1 25.1597,E2 452.425} C_DIS
LIN {X 87.523,Y -6.184,Z 88,A -10.1028,B 24.9183,C -2.0868,E1 25.1591,E2 455.1098} C_DIS
LIN {X 87.2099,Y -9.6515,Z 88,A -11.9075,B 24.9176,C -2.0958,E1 25.1586,E2 456.8827} C_DIS
LIN {X 86.8972,Y -12.139,Z 88,A -14.3832,B 24.9203,C -2.0615,E1 25.1576,E2 459.4247} C_DIS
LIN {X 86.1144,Y -16.817,Z 88,A -16.1571,B 24.9175,C -2.0976,E1 25.1568,E2 461.1029} C_DIS
LIN {X 84.6664,Y -23.0233,Z 88,A -21.4952,B 24.9217,C -2.0435,E1 25.1531,E2 466.5379} C_DIS
LIN {X 83.397,Y -27.2664,Z 88,A -23.7921,B 24.9208,C -2.0551,E1 25.1512,E2 468.7945} C_DIS
LIN {X 81.7818,Y -31.785,Z 88,A -26.6457,B 24.9208,C -2.0552,E1 25.1484,E2 471.6319} C_DIS
LIN {X 79.8257,Y -36.4208,Z 88,A -30.3911,B 24.9228,C -2.0293,E1 25.1442,E2 475.4179} C_DIS
LIN {X 78.422,Y -39.3525,Z 88,A -32.012,B 24.9219,C -2.0404,E1 25.1422,E2 477.004} C_DIS
LIN {X 76.4573,Y -43.0436,Z 88,A -34.896,B 24.9229,C -2.0271,E1 25.1384,E2 479.9043} C_DIS
LIN {X 74.6705,Y -46.0753,Z 88,A -36.9652,B 24.9229,C -2.0285,E1 25.1354,E2 481.9597} C_DIS
LIN {X 72.4044,Y -49.5605,Z 88,A -39.6689,B 24.9234,C -2.0213,E1 25.1312,E2 484.667} C_DIS
LIN {X 69.5904,Y -53.4382,Z 88,A -42.7002,B 24.9238,C -2.0162,E1 25.1262,E2 487.6958} C_DIS
LIN {X 65.707,Y -58.1488,Z 88,A -46.5942,B 24.9243,C -2.0089,E1 25.1193,E2 491.589} C_DIS
LIN {X 62.0974,Y -61.9885,Z 88,A -50.0261,B 24.9249,C -2.0007,E1 25.1127,E2 495.0253} C_DIS
LIN {X 57.9078,Y -65.9181,Z 88,A -53.5993,B 24.9251,C -1.998,E1 25.1054,E2 498.5904} C_DIS
LIN {X 54.1219,Y -69.0608,Z 88,A -56.9429,B 24.926,C -1.9864,E1 25.0981,E2 501.9487} C_DIS
LIN {X 49.3513,Y -72.5461,Z 88,A -60.9699,B 24.927,C -1.9727,E1 25.089,E2 505.994} C_DIS
LIN {X 46.8392,Y -74.1937,Z 88,A -63.1926,B 24.928,C -1.9601,E1 25.0837,E2 508.2391} C_DIS
LIN {X 42.6026,Y -76.704,Z 88,A -66.573,B 24.9288,C -1.9489,E1 25.0754,E2 511.636} C_DIS
LIN {X 39.5627,Y -78.3161,Z 88,A -69.128,B 24.9298,C -1.9349,E1 25.069,E2 514.2171} C_DIS
LIN {X 35.8671,Y -80.0752,Z 88,A -71.2778,B 24.9288,C -1.9481,E1 25.0636,E2 516.3303} C_DIS
LIN {X 31.4928,Y -81.8954,Z 88,A -74.1034,B 24.9285,C -1.9527,E1 25.0563,E2 519.1388} C_DIS
LIN {X 26.6293,Y -83.6032,Z 88,A -78.0886,B 24.9303,C -1.9282,E1 25.0457,E2 523.1742} C_DIS
LIN {X 23.1562,Y -84.6305,Z 88,A -79.8278,B 24.929,C -1.9461,E1 25.0411,E2 524.8681} C_DIS
LIN {X 18.7091,Y -85.7229,Z 88,A -83.1912,B 24.9301,C -1.9311,E1 25.0319,E2 528.2624} C_DIS
LIN {X 15.3158,Y -86.394,Z 88,A -85.9587,B 24.9314,C -1.9129,E1 25.0242,E2 531.0701} C_DIS
LIN {X 10.788,Y -87.0764,Z 88,A -88.1156,B 24.9296,C -1.9377,E1 25.0184,E2 533.1663} C_DIS
LIN {X 7.2581,Y -87.4405,Z 88,A -90.9734,B 24.9309,C -1.9192,E1 25.0103,E2 536.0665} C_DIS
LIN {X 3.6901,Y -87.6632,Z 88,A -92.969,B 24.9302,C -1.9291,E1 25.0048,E2 538.0379} C_DIS
LIN {X 0.5986,Y -87.7362,Z 88,A -94.4863,B 24.9291,C -1.9447,E1 25.0007,E2 539.518} C_DIS
Enddeposition()
LIN {X 0.5986,Y -87.7362,Z 88,A -94.4863,B 24.9291,C -1.9447,E1 25.0007,E2 539.518} C_DIS
Startdeposition()
$VEL.CP = VEL_PRINT
LIN {X 2.6644,Y -86.8188,Z 88,A -92.4777,B 24.9264,C -1.9812,E1 25.0065,E2 537.4233} C_DIS
LIN {X 6.3752,Y -86.6251,Z 88,A -89.6263,B 24.9254,C -1.9952,E1 25.0145,E2 534.5396} C_DIS
LIN {X 10.0146,Y -86.2805,Z 88,A -87.0593,B 24.9249,C -2.0017,E1 25.0217,E2 531.9591} C_DIS
LIN {X 13.2014,Y -85.8506,Z 88,A -85.0713,B 24.9251,C -1.9988,E1 25.0272,E2 529.9798} C_DIS
LIN {X 17.8274,Y -85.0113,Z 88,A -81.54,B 24.9238,C -2.0158,E1 25.0369,E2 526.4127} C_DIS
LIN {X 21.9225,Y -84.0482,Z 88,A -79.7218,B 24.926,C -1.9868,E1 25.0417,E2 524.6659} C_DIS
LIN {X 26.6072,Y -82.6842,Z 88,A -75.8736,B 24.9241,C -2.0114,E1 25.0521,E2 520.7662} C_DIS
LIN {X 30.1164,Y -81.4724,Z 88,A -73.8883,B 24.9251,C -1.9991,E1 25.0572,E2 518.8142} C_DIS
LIN {X 35.398,Y -79.3202,Z 88,A -69.6601,B 24.9235,C -2.0202,E1 25.0682,E2 514.546} C_DIS
LIN {X 38.3405,Y -77.9402,Z 88,A -68.3586,B 24.9254,C -1.9953,E1 25.0713,E2 513.307} C_DIS
LIN {X 41.8281,Y -76.1258,Z 88,A -65.1019,B 24.9233,C -2.0221,E1 25.0794,E2 509.9961} C_DIS
LIN {X 47.0589,Y -73.0075,Z 88,A -61.8549,B 24.9247,C -2.0034,E1 25.0871,E2 506.8033} C_DIS
LIN {X 48.7571,Y -71.8844,Z 88,A -59.5356,B 24.922,C -2.0394,E1 25.0926,E2 504.4069} C_DIS
LIN {X 51.5908,Y -69.8783,Z 88,A -57.7053,B 24.9229,C -2.0283,E1 25.0966,E2 502.6092} C_DIS
LIN {X 54.3467,Y -67.7574,Z 88,A -55.0185,B 24.9214,C -2.0468,E1 25.1026,E2 499.8887} C_DIS
LIN {X 56.9155,Y -65.615,Z 88,A -53.6578,B 24.9233,C -2.0227,E1 25.1054,E2 498.5904} C_DIS
LIN {X 60.7321,Y -62.0985,Z 88,A -49.9433,B 24.9219,C -2.0407,E1 25.113,E2 494.8485} C_DIS
LIN {X 64.6925,Y -57.9611,Z 88,A -46.652,B 24.9225,C -2.0333,E1 25.1193,E2 491.589} C_DIS
LIN {X 67.5371,Y -54.6201,Z 88,A -43.363,B 24.9209,C -2.0543,E1 25.1252,E2 488.2653} C_DIS
LIN {X 69.886,Y -51.5817,Z 88,A -40.575,B 24.9196,C -2.07,E1 25.13,E2 485.4536} C_DIS
LIN {X 71.5366,Y -49.2672,Z 88,A -38.7304,B 24.9193,C -2.0741,E1 25.1329,E2 483.6084} C_DIS
LIN {X 74.6562,Y -44.3973,Z 88,A -35.0763,B 24.9189,C -2.0792,E1 25.1383,E2 479.9606} C_DIS
LIN {X 76.9547,Y -40.2819,Z 88,A -32.4497,B 24.9195,C -2.0715,E1 25.1418,E2 477.3661} C_DIS
LIN {X 79.1997,Y -35.6653,Z 88,A -28.273,B 24.9166,C -2.1092,E1 25.1469,E2 473.1227} C_DIS
LIN {X 81.0799,Y -31.1582,Z 88,A -24.6054,B 24.9145,C -2.1348,E1 25.1507,E2 469.415} C_DIS
LIN {X 82.565,Y -26.9758,Z 88,A -22.2152,B 24.9153,C -2.1249,E1 25.1527,E2 467.0618} C_DIS
LIN {X 84.0073,Y -22.0819,Z 88,A -18.1143,B 24.9124,C -2.1616,E1 25.1557,E2 462.8978} C_DIS
LIN {X 85.1911,Y -16.9515,Z 88,A -15.4368,B 24.9138,C -2.1443,E1 25.1572,E2 460.2768} C_DIS
LIN {X 86.1758,Y -10.8816,Z 88,A -11.4172,B 24.9128,C -2.1559,E1 25.1588,E2 456.2534} C_DIS
LIN {X 86.6504,Y -6.029,Z 88,A -8.0821,B 24.9116,C -2.1705,E1 25.1596,E2 452.9037} C_DIS
LIN {X 86.8549,Y -1.0508,Z 88,A -5.1818,B 24.9119,C -2.1673,E1 25.1598,E2 450.0282} C_DIS
LIN {X 86.7593,Y 4.2022,Z 88,A -1.4021,B 24.9101,C -2.1894,E1 25.1594,E2 446.2187} C_DIS
LIN {X 86.3605,Y 9.3023,Z 88,A 1.5491,B 24.9104,C -2.1852,E1 25.1587,E2 443.295} C_DIS
LIN {X 85.5725,Y 14.9056,Z 88,A 5.6075,B 24.9085,C -2.2083,E1 25.1569,E2 439.2059} C_DIS
LIN {X 84.4217,Y 20.4353,Z 88,A 8.9018,B 24.9088,C -2.2046,E1 25.155,E2 435.9394} C_DIS
LIN {X 82.9478,Y 25.7735,Z 88,A 12.8361,B 24.9071,C -2.2255,E1 25.1519,E2 431.9784} C_DIS
LIN {X 81.4694,Y 30.1245,Z 88,A 15.5234,B 24.9074,C -2.2224,E1 25.1494,E2 429.3135} C_DIS
LIN {X 80.3187,Y 33.0702,Z 88,A 17.693,B 24.9066,C -2.2313,E1 25.1471,E2 427.1349} C_DIS
LIN {X 78.8737,Y 36.3818,Z 88,A 20.553,B 24.9046,C -2.2546,E1 25.1438,E2 424.2353} C_DIS
LIN {X 77.3855,Y 39.4474,Z 88,A 22.2359,B 24.9058,C -2.2412,E1 25.1417,E2 422.593} C_DIS
LIN {X 75.3472,Y 43.2136,Z 88,A 25.0516,B 24.9052,C -2.2485,E1 25.1379,E2 419.7747} C_DIS
LIN {X 73.5559,Y 46.1972,Z 88,A 27.337,B 24.9047,C -2.2542,E1 25.1346,E2 417.4877} C_DIS
LIN {X 71.7967,Y 48.8864,Z 88,A 29.4215,B 24.9043,C -2.2584,E1 25.1313,E2 415.4036} C_DIS
LIN {X 68.9581,Y 52.8153,Z 88,A 32.3686,B 24.9043,C -2.2576,E1 25.1265,E2 412.4724} C_DIS
LIN {X 66.4776,Y 55.9071,Z 88,A 35.0472,B 24.9037,C -2.2659,E1 25.1218,E2 409.7866} C_DIS
LIN {X 64.6229,Y 58.0385,Z 88,A 38.1439,B 24.8997,C -2.3123,E1 25.1158,E2 406.5939} C_DIS
LIN {X 61.0748,Y 61.7615,Z 88,A 39.9945,B 24.9036,C -2.2671,E1 25.1124,E2 404.8582} C_DIS
LIN {X 56.8051,Y 65.7114,Z 88,A 44.0922,B 24.9022,C -2.2834,E1 25.1039,E2 400.7384} C_DIS
LIN {X 54.7088,Y 67.4652,Z 88,A 46.4541,B 24.9003,C -2.3056,E1 25.0987,E2 398.3331} C_DIS
LIN {X 51.7517,Y 69.7613,Z 88,A 48.8394,B 24.9001,C -2.3071,E1 25.0934,E2 395.953} C_DIS
LIN {X 48.8174,Y 71.8435,Z 88,A 51.7246,B 24.8983,C -2.3281,E1 25.0867,E2 393.0276} C_DIS
LIN {X 45.1585,Y 74.1978,Z 88,A 54.0756,B 24.8994,C -2.3151,E1 25.0812,E2 390.7149} C_DIS
LIN {X 41.1997,Y 76.4673,Z 88,A 56.959,B 24.8994,C -2.315,E1 25.0741,E2 387.8402} C_DIS
LIN {X 38.2586,Y 77.9808,Z 88,A 59.4101,B 24.8984,C -2.3266,E1 25.0679,E2 385.3681} C_DIS
LIN {X 35.3591,Y 79.3377,Z 88,A 60.8713,B 24.9001,C -2.3076,E1 25.0644,E2 383.9555} C_DIS
LIN {X 30.6968,Y 81.2547,Z 88,A 64.1597,B 24.8999,C -2.3098,E1 25.0559,E2 380.6695} C_DIS
LIN {X 28.3342,Y 82.1096,Z 88,A 66.0092,B 24.8992,C -2.3174,E1 25.0509,E2 378.8056} C_DIS
LIN {X 25.4863,Y 83.0368,Z 88,A 68.1919,B 24.8985,C -2.3257,E1 25.0451,E2 376.6073} C_DIS
LIN {X 19.9495,Y 84.5387,Z 88,A 71.5121,B 24.8996,C -2.313,E1 25.0362,E2 373.3222} C_DIS
LIN {X 17.5842,Y 85.0612,Z 88,A 73.9255,B 24.8973,C -2.3399,E1 25.0294,E2 370.8481} C_DIS
LIN {X 14.1542,Y 85.6988,Z 88,A 75.3247,B 24.8997,C -2.3119,E1 25.0258,E2 369.5167} C_DIS
LIN {X 9.3696,Y 86.3535,Z 88,A 78.6399,B 24.8993,C -2.3167,E1 25.0166,E2 366.193} C_DIS
LIN {X 6.7181,Y 86.5997,Z 88,A 81.2022,B 24.8971,C -2.3423,E1 25.0093,E2 363.5712} C_DIS
LIN {X 3.0861,Y 86.8059,Z 88,A 82.966,B 24.8988,C -2.322,E1 25.0045,E2 361.8561} C_DIS
LIN {X -1.0648,Y 86.8548,Z 88,A 85.5597,B 24.8993,C -2.317,E1 24.9973,E2 359.2744} C_DIS
LIN {X -7.8315,Y 86.506,Z 88,A 89.8044,B 24.9,C -2.3084,E1 24.9855,E2 355.0491} C_DIS
LIN {X -12.5501,Y 85.9489,Z 88,A 93.3571,B 24.8991,C -2.3193,E1 24.9756,E2 351.4678} C_DIS
LIN {X -19.1644,Y 84.7201,Z 88,A 97.54,B 24.9001,C -2.3079,E1 24.9642,E2 347.3073} C_DIS
LIN {X -23.7159,Y 83.5593,Z 88,A 100.7656,B 24.9,C -2.3087,E1 24.9555,E2 344.0752} C_DIS
LIN {X -26.4018,Y 82.7507,Z 88,A 103.1124,B 24.8989,C -2.3216,E1 24.9491,E2 341.6936} C_DIS
LIN {X -31.1876,Y 81.0688,Z 88,A 105.9275,B 24.9006,C -2.3013,E1 24.9418,E2 338.9211} C_DIS
LIN {X -33.6186,Y 80.09,Z 88,A 108.6392,B 24.8983,C -2.3285,E1 24.9347,E2 336.1384} C_DIS
LIN {X -37.4543,Y 78.3697,Z 88,A 110.3499,B 24.9014,C -2.2924,E1 24.9305,E2 334.5095} C_DIS
LIN {X -42.0344,Y 76.0121,Z 88,A 114,B 24.9013,C -2.2942,E1 24.9215,E2 330.8451} C_DIS
LIN {X -45.7156,Y 73.8567,Z 88,A 117.0098,B 24.9012,C -2.2949,E1 24.9142,E2 327.8244} C_DIS
LIN {X -49.4372,Y 71.4185,Z 88,A 119.818,B 24.902,C -2.2854,E1 24.9078,E2 325.0293} C_DIS
LIN {X -54.2209,Y 67.8595,Z 88,A 124.8018,B 24.9,C -2.3082,E1 24.8966,E2 319.9731} C_DIS
LIN {X -57.9933,Y 64.6637,Z 88,A 126.9046,B 24.9036,C -2.2668,E1 24.8924,E2 317.9607} C_DIS
LIN {X -60.8074,Y 62.025,Z 88,A 129.7511,B 24.9034,C -2.2695,E1 24.8866,E2 315.0959} C_DIS
LIN {X -63.935,Y 58.7957,Z 88,A 132.9024,B 24.9035,C -2.2676,E1 24.8805,E2 311.9353} C_DIS
LIN {X -67.11,Y 55.144,Z 88,A 136.2909,B 24.9037,C -2.2651,E1 24.8744,E2 308.5372} C_DIS
LIN {X -69.1584,Y 52.5542,Z 88,A 137.7809,B 24.9059,C -2.2395,E1 24.872,E2 307.1014} C_DIS
LIN {X -71.9816,Y 48.6134,Z 88,A 140.9654,B 24.9067,C -2.2304,E1 24.8669,E2 303.9229} C_DIS
LIN {X -73.3498,Y 46.5255,Z 88,A 143.2529,B 24.9055,C -2.2441,E1 24.8634,E2 301.5911} C_DIS
LIN {X -76.2907,Y 41.5254,Z 88,A 146.5516,B 24.9077,C -2.218,E1 24.8589,E2 298.3375} C_DIS
LIN {X -77.5866,Y 39.0538,Z 88,A 149.9443,B 24.9044,C -2.2573,E1 24.8545,E2 294.8328} C_DIS
LIN {X -80.1172,Y 33.554,Z 88,A 152.6478,B 24.9085,C -2.2081,E1 24.8516,E2 292.2319} C_DIS
LIN {X -81.4082,Y 30.2913,Z 88,A 155.4053,B 24.9081,C -2.2136,E1 24.8489,E2 289.4457} C_DIS
LIN {X -83.127,Y 25.1943,Z 88,A 159.1696,B 24.9085,C -2.2087,E1 24.8457,E2 285.6713} C_DIS
LIN {X -84.1392,Y 21.5687,Z 88,A 160.5152,B 24.9118,C -2.1687,E1 24.8448,E2 284.4135} C_DIS
LIN {X -84.8447,Y 18.6009,Z 88,A 163.4349,B 24.9102,C -2.188,E1 24.8429,E2 281.4306} C_DIS
LIN {X -85.5024,Y 15.2956,Z 88,A 165.9239,B 24.9102,C -2.1885,E1 24.8417,E2 278.9256} C_DIS
LIN {X -86.0934,Y 11.5179,Z 88,A 167.515,B 24.913,C -2.154,E1 24.8411,E2 277.4075} C_DIS
LIN {X -86.5812,Y 6.9497,Z 88,A 171.4765,B 24.9116,C -2.1707,E1 24.8401,E2 273.3823} C_DIS
LIN {X -86.8012,Y 3.2272,Z 88,A 173.1444,B 24.9141,C -2.1403,E1 24.8399,E2 271.7769} C_DIS
LIN {X -86.8578,Y 0.6472,Z 88,A 175.7325,B 24.9125,C -2.1601,E1 24.8399,E2 269.126} C_DIS
LIN {X -86.8001,Y -3.2509,Z 88,A 178.416,B 24.9129,C -2.1551,E1 24.8401,E2 266.4383} C_DIS
LIN {X -86.5433,Y -7.4245,Z 88,A -179.7652,B 24.9157,C -2.1195,E1 24.8405,E2 264.6934} C_DIS
LIN {X -85.8201,Y -13.3987,Z 88,A -176.1764,B 24.9176,C -2.0963,E1 24.8417,E2 261.1386} C_DIS
LIN {X -85.2014,Y -16.8985,Z 88,A -173.1548,B 24.9167,C -2.1081,E1 24.8432,E2 258.0708} C_DIS
LIN {X -84.4882,Y -20.163,Z 88,A -171.0105,B 24.9173,C -2.0997,E1 24.8446,E2 255.9341} C_DIS
LIN {X -83.6708,Y -23.3224,Z 88,A -168.7964,B 24.9177,C -2.0949,E1 24.8462,E2 253.7185} C_DIS
LIN {X -82.6551,Y -26.6972,Z 88,A -165.492,B 24.916,C -2.1163,E1 24.8491,E2 250.344} C_DIS
LIN {X -81.0013,Y -31.3621,Z 88,A -163.4603,B 24.9196,C -2.0711,E1 24.851,E2 248.4088} C_DIS
LIN {X -79.1901,Y -35.6866,Z 88,A -159.8674,B 24.9191,C -2.0767,E1 24.8549,E2 244.7827} C_DIS
LIN {X -77.0905,Y -40.024,Z 88,A -156.8688,B 24.9202,C -2.0627,E1 24.8587,E2 241.8015} C_DIS
LIN {X -75.6013,Y -42.7702,Z 88,A -154.2346,B 24.9193,C -2.0739,E1 24.8623,E2 239.1268} C_DIS
LIN {X -73.8016,Y -45.8038,Z 88,A -152.8411,B 24.9219,C -2.0406,E1 24.8643,E2 237.8054} C_DIS
LIN {X -71.6696,Y -49.0738,Z 88,A -149.2111,B 24.92,C -2.0649,E1 24.87,E2 234.0993} C_DIS
LIN {X -69.4332,Y -52.1885,Z 88,A -147.5043,B 24.9224,C -2.0346,E1 24.8728,E2 232.4567} C_DIS
LIN {X -67.5376,Y -54.6195,Z 88,A -144.3232,B 24.9201,C -2.0638,E1 24.8785,E2 229.1912} C_DIS
LIN {X -64.3465,Y -58.3471,Z 88,A -142.2499,B 24.9233,C -2.0219,E1 24.8822,E2 227.2084} C_DIS
LIN {X -62.6026,Y -60.2123,Z 88,A -140.4158,B 24.9233,C -2.0227,E1 24.8857,E2 225.3644} C_DIS
LIN {X -59.1678,Y -63.5924,Z 88,A -137.375,B 24.9241,C -2.012,E1 24.8918,E2 222.3364} C_DIS
LIN {X -57.3447,Y -65.2401,Z 88,A -135.1886,B 24.9231,C -2.0257,E1 24.8964,E2 220.1086} C_DIS
LIN {X -54.5111,Y -67.6254,Z 88,A -132.9819,B 24.9239,C -2.0141,E1 24.9012,E2 217.9213} C_DIS
LIN {X -51.9466,Y -69.6149,Z 88,A -131.1687,B 24.925,C -2.0005,E1 24.9051,E2 216.1339} C_DIS
LIN {X -48.4583,Y -72.0858,Z 88,A -127.3587,B 24.923,C -2.026,E1 24.9141,E2 212.2505} C_DIS
LIN {X -44.9972,Y -74.2958,Z 88,A -125.5869,B 24.9255,C -1.9933,E1 24.9181,E2 210.5507} C_DIS
LIN {X -41.1985,Y -76.468,Z 88,A -122.0094,B 24.9242,C -2.0105,E1 24.927,E2 206.922} C_DIS
LIN {X -38.3168,Y -77.952,Z 88,A -120.6203,B 24.9261,C -1.9849,E1 24.9303,E2 205.5902} C_DIS
LIN {X -35.771,Y -79.1521,Z 88,A -118.5187,B 24.9257,C -1.9903,E1 24.9357,E2 203.4704} C_DIS
LIN {X -33.7076,Y -80.0525,Z 88,A -116.7325,B 24.9251,C -1.9981,E1 24.9403,E2 201.6617} C_DIS
LIN {X -29.7529,Y -81.605,Z 88,A -114.1393,B 24.9258,C -1.989,E1 24.947,E2 199.0847} C_DIS
LIN {X -22.8655,Y -83.7963,Z 88,A -109.7886,B 24.9271,C -1.9725,E1 24.9586,E2 194.7657} C_DIS
LIN {X -18.5992,Y -84.8451,Z 88,A -106.3759,B 24.926,C -1.9871,E1 24.9679,E2 191.3136} C_DIS
LIN {X -12.6923,Y -85.9287,Z 88,A -102.5015,B 24.9263,C -1.9831,E1 24.9786,E2 187.445} C_DIS
LIN {X -9.5034,Y -86.3395,Z 88,A -99.922,B 24.9252,C -1.9974,E1 24.9858,E2 184.8298} C_DIS
LIN {X -6.2338,Y -86.6365,Z 88,A -98.1889,B 24.9262,C -1.9835,E1 24.9906,E2 183.129} C_DIS
LIN {X -2.9153,Y -86.8111,Z 88,A -96.0921,B 24.9264,C -1.9807,E1 24.9964,E2 181.0384} C_DIS
LIN {X 0.5833,Y -86.8551,Z 88,A -93.7003,B 24.9262,C -1.984,E1 25.0031,E2 178.639} C_DIS
Enddeposition()
LIN {X 0.5833,Y -86.8551,Z 88,A -93.7003,B 24.9262,C -1.984,E1 25.0031,E2 178.639} C_DIS
Startdeposition()
$VEL.CP = VEL_PRINT
LIN {X 0.1576,Y -85.9792,Z 88,A -95.1526,B 24.9278,C -1.962,E1 24.9989,E2 180.1432} C_DIS
LIN {X -4.605,Y -85.8553,Z 88,A -98.1331,B 24.9274,C -1.9677,E1 24.9906,E2 183.1107} C_DIS
LIN {X -9.7525,Y -85.4241,Z 88,A -101.7099,B 24.9277,C -1.9637,E1 24.9807,E2 186.6988} C_DIS
LIN {X -15.6385,Y -84.5455,Z 88,A -105.4573,B 24.9271,C -1.9715,E1 24.9704,E2 190.431} C_DIS
LIN {X -19.7024,Y -83.6915,Z 88,A -108.5184,B 24.9277,C -1.9638,E1 24.9619,E2 193.5143} C_DIS
LIN {X -23.1916,Y -82.7921,Z 88,A -111.709,B 24.9293,C -1.9416,E1 24.9532,E2 196.7627} C_DIS
LIN {X -27.3734,Y -81.5048,Z 88,A -113.6991,B 24.9271,C -1.9715,E1 24.9481,E2 198.6851} C_DIS
LIN {X -30.3509,Y -80.4435,Z 88,A -115.7705,B 24.9269,C -1.9744,E1 24.9427,E2 200.7538} C_DIS
LIN {X -32.507,Y -79.5966,Z 88,A -117.5528,B 24.9273,C -1.9688,E1 24.938,E2 202.5534} C_DIS
LIN {X -35.5331,Y -78.2928,Z 88,A -119.6144,B 24.9269,C -1.9752,E1 24.9328,E2 204.6048} C_DIS
LIN {X -39.8347,Y -76.1943,Z 88,A -122.7485,B 24.9264,C -1.9807,E1 24.925,E2 207.734} C_DIS
LIN {X -43.3741,Y -74.2374,Z 88,A -125.4518,B 24.9262,C -1.9842,E1 24.9184,E2 210.437} C_DIS
LIN {X -46.7527,Y -72.157,Z 88,A -128.4544,B 24.9267,C -1.9777,E1 24.9112,E2 213.4647} C_DIS
LIN {X -50.7914,Y -69.3726,Z 88,A -131.3019,B 24.9253,C -1.9954,E1 24.9048,E2 216.2798} C_DIS
LIN {X -53.8018,Y -67.0661,Z 88,A -134.0135,B 24.9254,C -1.9945,E1 24.8988,E2 219.0034} C_DIS
LIN {X -56.7126,Y -64.6223,Z 88,A -136.6065,B 24.9252,C -1.9976,E1 24.8933,E2 221.599} C_DIS
LIN {X -60.029,Y -61.5555,Z 88,A -139.6127,B 24.9247,C -2.0038,E1 24.8872,E2 224.6028} C_DIS
LIN {X -62.3868,Y -59.1636,Z 88,A -141.86,B 24.9244,C -2.0084,E1 24.8828,E2 226.849} C_DIS
LIN {X -64.5175,Y -56.8326,Z 88,A -144.6454,B 24.9255,C -1.9938,E1 24.8776,E2 229.6816} C_DIS
LIN {X -67.0291,Y -53.8475,Z 88,A -146.4943,B 24.9234,C -2.0211,E1 24.8744,E2 231.4741} C_DIS
LIN {X -68.5034,Y -51.9592,Z 88,A -149.2711,B 24.9256,C -1.9918,E1 24.8697,E2 234.3339} C_DIS
LIN {X -71.5264,Y -47.7127,Z 88,A -151.6751,B 24.9227,C -2.0304,E1 24.866,E2 236.6579} C_DIS
LIN {X -73.2404,Y -45.0355,Z 88,A -154.2241,B 24.9232,C -2.0239,E1 24.8622,E2 239.2355} C_DIS
LIN {X -75.631,Y -40.8935,Z 88,A -156.9881,B 24.9216,C -2.0442,E1 24.8585,E2 241.9655} C_DIS
LIN {X -77.3396,Y -37.5638,Z 88,A -160.2476,B 24.9227,C -2.0299,E1 24.8544,E2 245.2767} C_DIS
LIN {X -79.0043,Y -33.921,Z 88,A -162.1814,B 24.9206,C -2.0578,E1 24.8523,E2 247.1546} C_DIS
LIN {X -80.7456,Y -29.5376,Z 88,A -165.9658,B 24.9213,C -2.0492,E1 24.8485,E2 250.9807} C_DIS
LIN {X -81.9312,Y -26.0724,Z 88,A -167.8502,B 24.9195,C -2.0718,E1 24.8469,E2 252.8221} C_DIS
LIN {X -82.9086,Y -22.773,Z 88,A -170.1534,B 24.919,C -2.0784,E1 24.8451,E2 255.1228} C_DIS
LIN {X -83.7261,Y -19.5524,Z 88,A -172.3319,B 24.9184,C -2.0861,E1 24.8437,E2 257.2957} C_DIS
LIN {X -84.5261,Y -15.745,Z 88,A -175.1886,B 24.9184,C -2.0869,E1 24.8421,E2 260.1674} C_DIS
LIN {X -84.9738,Y -13.1065,Z 88,A -177.3445,B 24.9187,C -2.0823,E1 24.8412,E2 262.347} C_DIS
LIN {X -85.4496,Y -9.5342,Z 88,A -179.1535,B 24.9168,C -2.106,E1 24.8406,E2 264.1103} C_DIS
LIN {X -85.725,Y -6.6031,Z 88,A 178.3842,B 24.9174,C -2.0986,E1 24.8401,E2 266.6052} C_DIS
LIN {X -85.9766,Y -0.6852,Z 88,A 174.8729,B 24.9155,C -2.123,E1 24.8398,E2 270.0792} C_DIS
LIN {X -85.9309,Y 2.8745,Z 88,A 172.6387,B 24.9146,C -2.1344,E1 24.8399,E2 272.2997} C_DIS
LIN {X -85.6933,Y 6.9995,Z 88,A 169.5871,B 24.9146,C -2.1351,E1 24.8405,E2 275.3681} C_DIS
LIN {X -85.293,Y 10.838,Z 88,A 167.5083,B 24.9128,C -2.1568,E1 24.8411,E2 277.4075} C_DIS
LIN {X -84.7221,Y 14.6534,Z 88,A 164.4642,B 24.9131,C -2.152,E1 24.8424,E2 280.4812} C_DIS
LIN {X -83.9008,Y 18.7909,Z 88,A 161.5477,B 24.9127,C -2.158,E1 24.8441,E2 283.4005} C_DIS
LIN {X -82.1691,Y 25.3097,Z 88,A 157.2724,B 24.911,C -2.1781,E1 24.8473,E2 287.6526} C_DIS
LIN {X -79.8868,Y 31.7894,Z 88,A 152.8655,B 24.9095,C -2.1968,E1 24.8514,E2 292.0398} C_DIS
LIN {X -78.3906,Y 35.3161,Z 88,A 149.3781,B 24.9109,C -2.1789,E1 24.8554,E2 295.5892} C_DIS
LIN {X -76.7996,Y 38.6577,Z 88,A 147.408,B 24.9092,C -2.1997,E1 24.8578,E2 297.5202} C_DIS
LIN {X -75.4829,Y 41.1666,Z 88,A 144.753,B 24.9105,C -2.1843,E1 24.8614,E2 300.2261} C_DIS
LIN {X -73.2657,Y 44.9956,Z 88,A 142.5785,B 24.9081,C -2.2138,E1 24.8645,E2 302.3414} C_DIS
LIN {X -71.5463,Y 47.6826,Z 88,A 140.701,B 24.907,C -2.2266,E1 24.8673,E2 304.1978} C_DIS
LIN {X -69.1496,Y 51.0959,Z 88,A 137.6943,B 24.9069,C -2.2278,E1 24.8722,E2 307.2163} C_DIS
LIN {X -66.1637,Y 54.9062,Z 88,A 134.5211,B 24.9061,C -2.2377,E1 24.8777,E2 310.3806} C_DIS
LIN {X -63.2503,Y 58.2374,Z 88,A 131.4492,B 24.9057,C -2.2417,E1 24.8834,E2 313.4568} C_DIS
LIN {X -60.5862,Y 61.0039,Z 88,A 128.5456,B 24.906,C -2.2383,E1 24.8892,E2 316.3809} C_DIS
LIN {X -57.5486,Y 63.8791,Z 88,A 125.2889,B 24.9066,C -2.2316,E1 24.896,E2 319.6666} C_DIS
LIN {X -54.2732,Y 66.6841,Z 88,A 122.7026,B 24.9054,C -2.2458,E1 24.9015,E2 322.2288} C_DIS
LIN {X -51.6361,Y 68.7462,Z 88,A 121.0971,B 24.9035,C -2.2682,E1 24.9049,E2 323.787} C_DIS
LIN {X -49.2626,Y 70.4668,Z 88,A 119.0829,B 24.9033,C -2.2704,E1 24.9095,E2 325.8028} C_DIS
LIN {X -45.2162,Y 73.1298,Z 88,A 115.6373,B 24.9033,C -2.2702,E1 24.9176,E2 329.2598} C_DIS
LIN {X -41.988,Y 75.0289,Z 88,A 112.7157,B 24.904,C -2.2625,E1 24.9248,E2 332.2085} C_DIS
LIN {X -38.9142,Y 76.6684,Z 88,A 111.0825,B 24.902,C -2.286,E1 24.9287,E2 333.7901} C_DIS
LIN {X -35.8201,Y 78.162,Z 88,A 108.2714,B 24.9029,C -2.2745,E1 24.9359,E2 336.6357} C_DIS
LIN {X -31.9239,Y 79.8338,Z 88,A 105.8202,B 24.9017,C -2.2892,E1 24.9422,E2 339.0573} C_DIS
LIN {X -28.9726,Y 80.9517,Z 88,A 103.4964,B 24.902,C -2.2855,E1 24.9483,E2 341.3947} C_DIS
LIN {X -25.2416,Y 82.1902,Z 88,A 101.0742,B 24.9012,C -2.2943,E1 24.9547,E2 343.8002} C_DIS
LIN {X -23.1001,Y 82.818,Z 88,A 99.1412,B 24.9022,C -2.2828,E1 24.96,E2 345.7637} C_DIS
LIN {X -19.1866,Y 83.8106,Z 88,A 96.1541,B 24.9028,C -2.2766,E1 24.9682,E2 348.7696} C_DIS
LIN {X -15.2333,Y 84.6183,Z 88,A 94.3124,B 24.9004,C -2.3037,E1 24.9731,E2 350.5488} C_DIS
LIN {X -12.2187,Y 85.106,Z 88,A 91.5723,B 24.9021,C -2.2841,E1 24.9808,E2 353.3378} C_DIS
LIN {X -8.6652,Y 85.5413,Z 88,A 89.9647,B 24.9,C -2.3086,E1 24.9851,E2 354.8881} C_DIS
LIN {X -2.9268,Y 85.9292,Z 88,A 84.9404,B 24.903,C -2.2743,E1 24.9993,E2 359.9952} C_DIS
LIN {X 1.9528,Y 85.9572,Z 88,A 82.9765,B 24.8996,C -2.3136,E1 25.0045,E2 361.8655} C_DIS
LIN {X 7.076,Y 85.6872,Z 88,A 79.4535,B 24.8998,C -2.3104,E1 25.0144,E2 365.3947} C_DIS
LIN {X 10.5254,Y 85.3317,Z 88,A 76.8363,B 24.9007,C -2.3007,E1 25.0217,E2 368.0333} C_DIS
LIN {X 13.2634,Y 84.9495,Z 88,A 74.6083,B 24.9018,C -2.2883,E1 25.0279,E2 370.2885} C_DIS
LIN {X 16.5206,Y 84.3769,Z 88,A 73.0114,B 24.9002,C -2.3061,E1 25.0322,E2 371.8414} C_DIS
LIN {X 19.3304,Y 83.7774,Z 88,A 71.2196,B 24.9,C -2.309,E1 25.037,E2 373.6239} C_DIS
LIN {X 22.6934,Y 82.9301,Z 88,A 68.6297,B 24.9008,C -2.2988,E1 25.0441,E2 376.2339} C_DIS
LIN {X 26.0502,Y 81.9384,Z 88,A 66.3882,B 24.9008,C -2.2999,E1 25.05,E2 378.4687} C_DIS
LIN {X 28.6292,Y 81.0723,Z 88,A 64.7033,B 24.9005,C -2.3024,E1 25.0545,E2 380.1444} C_DIS
LIN {X 30.9894,Y 80.201,Z 88,A 62.4704,B 24.9022,C -2.2833,E1 25.0604,E2 382.4179} C_DIS
LIN {X 34.5305,Y 78.7401,Z 88,A 59.7892,B 24.9028,C -2.2765,E1 25.0673,E2 385.1087} C_DIS
LIN {X 37.6871,Y 77.2803,Z 88,A 57.6161,B 24.9026,C -2.2782,E1 25.0727,E2 387.272} C_DIS
LIN {X 41.8279,Y 75.1183,Z 88,A 55.3671,B 24.9006,C -2.3017,E1 25.0781,E2 389.4589} C_DIS
LIN {X 45.4931,Y 72.9567,Z 88,A 51.615,B 24.9035,C -2.2681,E1 25.0873,E2 393.279} C_DIS
LIN {X 48.1778,Y 71.2125,Z 88,A 50.2819,B 24.9016,C -2.2904,E1 25.0902,E2 394.5547} C_DIS
LIN {X 50.5054,Y 69.582,Z 88,A 48.048,B 24.9028,C -2.2762,E1 25.0954,E2 396.8146} C_DIS
LIN {X 53.9012,Y 66.9856,Z 88,A 45.2198,B 24.9032,C -2.2717,E1 25.1016,E2 399.643} C_DIS
LIN {X 58.8951,Y 62.6394,Z 88,A 40.9109,B 24.9036,C -2.2664,E1 25.1106,E2 403.9474} C_DIS
LIN {X 61.2363,Y 60.3527,Z 88,A 37.7925,B 24.9066,C -2.2311,E1 25.1168,E2 407.1358} C_DIS
LIN {X 64.3492,Y 57.0235,Z 88,A 35.6083,B 24.9048,C -2.2522,E1 25.1208,E2 409.2604} C_DIS
LIN {X 67.2105,Y 53.6211,Z 88,A 32.9747,B 24.9045,C -2.2562,E1 25.1255,E2 411.8724} C_DIS
LIN {X 68.8232,Y 51.5335,Z 88,A 30.6401,B 24.9065,C -2.2328,E1 25.1295,E2 414.2512} C_DIS
LIN {X 71.3375,Y 47.9932,Z 88,A 28.0037,B 24.9064,C -2.2341,E1 25.1336,E2 416.8716} C_DIS
LIN {X 73.2799,Y 44.9724,Z 88,A 25.665,B 24.9067,C -2.2297,E1 25.1371,E2 419.2089} C_DIS
LIN {X 74.7642,Y 42.4596,Z 88,A 23.1561,B 24.9087,C -2.2057,E1 25.1406,E2 421.7616} C_DIS
LIN {X 76.4726,Y 39.2976,Z 88,A 20.6843,B 24.9095,C -2.1966,E1 25.1438,E2 424.2418} C_DIS
LIN {X 78.2062,Y 35.7253,Z 88,A 18.7523,B 24.9081,C -2.213,E1 25.146,E2 426.1245} C_DIS
LIN {X 79.3802,Y 33.0341,Z 88,A 16.817,B 24.9085,C -2.2081,E1 25.1481,E2 428.0607} C_DIS
LIN {X 80.4111,Y 30.4365,Z 88,A 15.0984,B 24.9085,C -2.2076,E1 25.1499,E2 429.7711} C_DIS
LIN {X 81.3139,Y 27.9393,Z 88,A 12.935,B 24.9101,C -2.189,E1 25.1519,E2 431.9661} C_DIS
LIN {X 82.8966,Y 22.8175,Z 88,A 9.6197,B 24.9103,C -2.187,E1 25.1545,E2 435.2673} C_DIS
LIN {X 83.7442,Y 19.4741,Z 88,A 6.4858,B 24.9132,C -2.1518,E1 25.1565,E2 438.4662} C_DIS
LIN {X 84.6538,Y 15.0364,Z 88,A 4.8315,B 24.9101,C -2.1887,E1 25.1574,E2 440.0237} C_DIS
LIN {X 85.3676,Y 10.2347,Z 88,A 1.1872,B 24.9121,C -2.1645,E1 25.1588,E2 443.7037} C_DIS
LIN {X 85.6124,Y 7.9265,Z 88,A -1.0184,B 24.9143,C -2.1372,E1 25.1594,E2 445.9606} C_DIS
LIN {X 85.8799,Y 4.144,Z 88,A -3.6612,B 24.9153,C -2.1252,E1 25.1597,E2 448.6158} C_DIS
LIN {X 85.9796,Y -0.018,Z 88,A -5.68,B 24.9139,C -2.142,E1 25.1597,E2 450.5832} C_DIS
LIN {X 85.7777,Y -5.8739,Z 88,A -9.3514,B 24.9143,C -2.1375,E1 25.1594,E2 454.2433} C_DIS
LIN {X 85.4483,Y -9.545,Z 88,A -11.9699,B 24.9154,C -2.124,E1 25.1586,E2 456.8781} C_DIS
LIN {X 85.1735,Y -11.7435,Z 88,A -14.3835,B 24.9183,C -2.0875,E1 25.1577,E2 459.3637} C_DIS
LIN {X 84.3949,Y -16.4271,Z 88,A -16.3332,B 24.9158,C -2.1187,E1 25.1567,E2 461.2284} C_DIS
LIN {X 83.3397,Y -21.1398,Z 88,A -19.7476,B 24.9172,C -2.1018,E1 25.1546,E2 464.6629} C_DIS
LIN {X 82.4915,Y -24.2387,Z 88,A -21.8303,B 24.9175,C -2.097,E1 25.153,E2 466.7448} C_DIS
Enddeposition()
END
